Yaskawa INFORM job: X2_8A-21A(90,0).JBI

/JOB
//NAME X2_8A-21A(90,0)
///FOLDERNAME X2
//POS
///NPOS 910,910,910,41,0,0
///TOOL 0
///POSTYPE PULSE
///PULSE
C00000=12667,-135547,-130714,-31270,45596,0
C00001=9315,-159766,-119262,3212,6219,-55552
C00002=157761,-135547,-130714,-31270,45596,69143
C00003=154472,-113934,-104337,-41712,51336,70449
C00004=149832,-108771,-100172,-39130,49259,68869
C00005=148058,-106656,-98467,-38074,48499,68236
C00006=148062,-106275,-96666,-38578,47777,68578
C00007=148058,-106656,-98467,-38074,48499,68236
C00008=147997,-106381,-96958,-38469,47847,68508
C00009=145894,-104035,-96109,-36815,47477,67498
C00010=147997,-106381,-96958,-38469,47847,68508
C00011=154410,-113635,-102825,-42095,50721,70729
C00012=154342,-120637,-107041,-25827,48602,38771
C00013=150292,-111683,-102360,-22573,48994,36710
C00014=148798,-108210,-100464,-21373,49171,35962
C00015=146664,-105787,-99597,-19708,49308,34937
C00016=146949,-106220,-99797,-19932,49282,35074
C00017=147721,-103636,-97533,-20478,49410,35405
C00018=146949,-106220,-99797,-19932,49282,35074
C00019=152261,-118724,-106469,-24248,48548,37770
C00020=148295,-114597,-117137,6490,60568,69086
C00021=147868,-109631,-111600,6790,59752,68875
C00022=147704,-107727,-109395,6911,59390,68790
C00023=147708,-107860,-107783,6984,58336,68724
C00024=147704,-107727,-109395,6911,59390,68790
C00025=147723,-107760,-107968,6963,58499,68740
C00026=147306,-102596,-106094,7098,60024,68678
C00027=147723,-107760,-107968,6963,58499,68740
C00028=148315,-114751,-115749,6537,59639,69038
C00029=148355,-114889,-117236,6461,60467,69101
C00030=147925,-109892,-111692,6763,59663,68890
C00031=147761,-107977,-109485,6884,59305,68805
C00032=147764,-108104,-107870,6957,58254,68739
C00033=147777,-108153,-108078,6942,58354,68751
C00034=147358,-102980,-106206,7078,59886,68688
C00035=147777,-108153,-108078,6942,58354,68751
C00036=148373,-115211,-115873,6515,59468,69049
C00037=147696,-122269,-111871,35505,39043,51945
C00038=147690,-118447,-100224,39719,34874,49579
C00039=148491,-109409,-94254,38171,35277,50420
C00040=148787,-105724,-91002,38010,35060,50504
C00041=148789,-105382,-89977,38411,34697,50285
C00042=149058,-101689,-89016,37046,35623,51030
C00043=149145,-100783,-88679,36755,35795,51189
C00044=149058,-101689,-89016,37046,35623,51030
C00045=145777,-99657,-88811,39022,37803,49998
C00046=148139,-100407,-89095,37251,36591,50936
C00047=145777,-99657,-88811,39022,37803,49998
C00048=147690,-118447,-100224,39719,34874,49579
C00049=128033,-128545,-103748,39689,32513,43973
C00050=128383,-118409,-97778,37905,33566,44930
C00051=128511,-114277,-94563,37658,33626,45064
C00052=128512,-113804,-93446,38069,33271,44843
C00053=129119,-111006,-93029,36452,33958,45715
C00054=129434,-109852,-92636,35862,34111,46033
C00055=128358,-113721,-93936,37885,33613,44941
C00056=176216,-70111,-78093,-55162,70856,80763
C00057=174311,-70781,-78417,-54616,69674,80426
C00058=176216,-70111,-78093,-55162,70856,80763
C00059=181747,-69996,-81392,-56304,75271,81045
C00060=178033,-77165,-93769,-42680,75059,77098
C00061=164745,-109340,-116699,3009,62053,68278
C00062=145851,-112599,-102075,47717,41998,56322
C00063=148044,-104803,-96379,45883,41204,57334
C00064=148864,-101708,-93474,45490,40644,57533
C00065=148866,-101457,-92299,45986,40221,57239
C00066=148863,-101834,-94104,45225,40876,57690
C00067=145127,-99228,-91361,47944,42572,56214
C00068=147466,-100038,-91670,46636,41186,56907
C00069=145127,-99228,-91361,47944,42572,56214
C00070=146129,-107372,-95667,48598,40993,55782
C00071=148216,-109089,-93488,49289,38371,55335
C00072=148344,-107837,-93052,48851,38553,55585
C00073=147906,-112054,-94498,50363,37947,54724
C00074=145851,-112599,-102075,47717,41998,56322
C00075=158250,-140903,-124067,47621,67451,49320
C00076=161740,-133075,-117656,46661,65672,50232
C00077=162335,-130592,-114553,46699,64919,50156
C00078=162276,-129951,-113381,46845,64676,49998
C00079=160420,-132544,-115533,47350,65644,49520
C00080=135901,-74424,-73697,74364,100921,31256
C00081=137788,-75503,-74147,74218,99532,31324
C00082=138769,-76027,-74362,74146,98812,31363
C00083=135901,-74424,-73697,74364,100921,31256
C00084=149282,-147643,-98518,79858,51263,26133
C00085=149394,-146891,-98381,79629,51249,26315
C00086=148448,-152811,-99407,81432,51428,24854
C00087=139735,-166147,-105854,82069,56849,22658
C00088=180438,-97574,-115199,33764,102267,-52414
C00089=189965,-108899,-115705,31971,94091,-51156
C00090=189186,-107218,-114531,32087,94499,-51341
C00091=189186,-107583,-113435,32037,93763,-51550
C00092=190629,-109833,-115910,31859,93547,-51055
C00093=186867,-102382,-113240,32521,96788,-51574
C00094=187005,-102964,-110979,32373,95300,-51952
C00095=188888,-106610,-112304,32065,93703,-51681
C00096=187005,-102964,-110979,32373,95300,-51952
C00097=188021,-107681,-112675,32159,93748,-52003
C00098=189590,-103281,-111094,32025,94271,-51250
C00099=188021,-107681,-112675,32159,93748,-52003
C00100=180438,-97574,-115199,33764,102267,-52414
C00101=185735,-83978,-109774,33564,103394,-50026
C00102=199988,-77820,-108712,-11582,98175,38155
C00103=204749,-56978,-92496,-29836,109182,47433
C00104=202460,-56662,-91339,-29422,107990,46925
C00105=201413,-57385,-91726,-29256,107546,46663
C00106=201611,-57041,-91542,-29296,107663,46703
C00107=201611,-58240,-90431,-29070,106521,47008
C00108=203359,-50274,-87822,-29763,109247,46906
C00109=195470,-25798,-72981,-29209,109868,43903
C00110=195013,-27562,-73704,-29036,109327,43888
C00111=194283,-28250,-74172,-28893,109053,43704
C00112=194480,-28066,-74047,-28932,109127,43754
C00113=194480,-29296,-73135,-28708,108075,44034
C00114=195605,-24849,-71507,-29147,109538,44038
C00115=191110,-5546,-57842,-28597,109561,42465
C00116=192519,-3768,-54500,-33008,111368,41387
C00117=191992,-5303,-55742,-32912,111174,41254
C00118=192059,-5108,-55586,-32924,111198,41271
C00119=192059,-6294,-54683,-32651,110210,41583
C00120=192882,-2296,-53893,-33162,111810,41382
C00121=203365,-15491,-64400,-34648,115083,44256
C00122=218411,-26661,-75493,-58573,107247,46176
C00123=145332,-87800,-123084,-4045,108310,-15756
C00124=109199,-104290,-129101,21867,105305,-43874
C00125=112610,-115777,-129409,14908,94573,-36374
C00126=117115,-112620,-124614,14006,92529,-35127
C00127=118008,-112320,-123068,13816,91609,-34934
C00128=118007,-112900,-122267,13806,90840,-35020
C00129=118044,-112536,-122505,13803,91159,-34973
C00130=118576,-105776,-120168,13731,93052,-34586
C00131=118044,-112536,-122505,13803,91159,-34973
C00132=125955,-111499,-122045,12179,90192,-32457
C00133=127333,-111877,-122174,11884,89885,-32033
C00134=124755,-111115,-121914,12435,90480,-32824
C00135=119624,-116552,-128230,13509,92325,-34321
C00136=117231,-121833,-124467,22052,85463,-28755
C00137=122341,-114124,-118662,20866,84531,-27121
C00138=123318,-113111,-117155,20643,83910,-26885
C00139=123641,-113323,-116249,20585,83205,-26892
C00140=123595,-112804,-116375,20585,83540,-26851
C00141=123397,-106736,-114247,20589,85286,-26623
C00142=123595,-112804,-116375,20585,83540,-26851
C00143=116023,-114044,-115764,22346,84523,-29358
C00144=117346,-116777,-115957,22098,82979,-29171
C00145=118867,-116723,-116143,21757,82713,-28674
C00146=116293,-116772,-115815,22329,83179,-29512
C00147=117231,-121833,-124467,22052,85463,-28755
C00148=154726,-134692,-133300,-19029,79240,-32627
C00149=155157,-123239,-125350,-19102,80279,-32639
C00150=155214,-122106,-123677,-19140,79867,-32554
C00151=155216,-122330,-122794,-19175,79245,-32454
C00152=155272,-122641,-123186,-19186,79334,-32449
C00153=154565,-115790,-120970,-18882,81218,-32994
C00154=155272,-122449,-123985,-19155,79894,-32538
C00155=110972,-119209,-121408,15853,79302,-48266
C00156=109086,-133769,-122042,16854,72857,-49812
C00157=111848,-135958,-122676,16103,71595,-48979
C00158=109086,-133769,-122042,16854,72857,-49812
C00159=108592,-130707,-130810,16554,79646,-49045
C00160=120610,-122471,-119242,21572,81234,-22537
C00161=120610,-122484,-118172,21604,80613,-22649
C00162=120610,-122391,-116483,21658,79689,-22817
C00163=120610,-122419,-116833,21647,79876,-22783
C00164=120610,-122423,-116832,21647,79874,-22783
C00165=120610,-122419,-116833,21647,79876,-22783
C00166=120610,-122416,-116761,21649,79836,-22790
C00167=120610,-122436,-116768,21650,79830,-22791
C00168=120610,-122416,-116761,21649,79836,-22790
C00169=120611,-122370,-120508,21535,82009,-22397
C00170=120611,-120494,-126735,3133,87635,-4471
C00171=120611,-121772,-123926,3138,85252,-4531
C00172=120611,-122092,-122744,3141,84362,-4553
C00173=120611,-122362,-121169,3146,83256,-4581
C00174=120611,-122286,-121724,3144,83636,-4571
C00175=120611,-122290,-121724,3144,83633,-4571
C00176=120611,-122286,-121724,3144,83636,-4571
C00177=120611,-121006,-125813,3134,86805,-4492
C00178=120621,-120378,-125991,12397,109990,-35253
C00179=136832,-143297,-133894,19017,104291,-40845
C00180=187686,-122249,-118318,34521,102174,-42234
C00181=187703,-122088,-115580,34298,100833,-42653
C00182=187707,-122010,-114917,34250,100525,-42749
C00183=187713,-121734,-113169,34135,99743,-42991
C00184=187707,-122010,-114917,34250,100525,-42749
C00185=187770,-121697,-112491,32279,113674,-44764
C00186=187767,-121692,-112491,32279,113678,-44765
C00187=187770,-121697,-112491,32279,113674,-44764
C00188=187667,-121438,-112064,34928,84963,-41689
C00189=187673,-121448,-112068,34927,84958,-41688
C00190=187667,-121438,-112064,34928,84963,-41689
C00191=187641,-121957,-115421,34884,86463,-41227
C00192=173591,-141106,-131528,9997,106250,-69327
C00193=160878,-120510,-126471,37,121976,-81968
C00194=160881,-121699,-123664,37,119637,-81967
C00195=160883,-121991,-122485,37,118762,-81967
C00196=160886,-122244,-120905,37,117660,-81966
C00197=160884,-122111,-121864,37,118318,-81967
C00198=160882,-122100,-121862,36,118322,-81968
C00199=160884,-122111,-121864,37,118318,-81967
C00200=160879,-120821,-125908,37,121469,-81968
C00201=160879,-120821,-131564,37,121469,-81968
C00202=126581,-129511,-133446,-8167,112012,-37796
C00203=82387,-124374,-130385,-21792,102809,55833
C00204=37550,-124758,-124791,-27166,84975,54517
C00205=35933,-124831,-122904,-26864,83389,54284
C00206=35589,-124875,-121597,-26827,82538,54351
C00207=35584,-124889,-121174,-26839,82296,54405
C00208=35764,-126387,-121953,-26892,82093,54519
C00209=31633,-125451,-121673,-25972,81076,53208
C00210=35764,-126387,-121953,-26892,82093,54519
C00211=46981,-157328,-126723,-35790,81436,33730
C00212=42905,-153934,-122174,-35701,78867,32870
C00213=42758,-143813,-119569,-35389,81762,31868
C00214=42905,-153934,-122174,-35701,78867,32870
C00215=53188,-117519,-120731,-36414,97747,30962
C00216=95179,-109851,-129540,-3422,106316,-17944
C00217=143691,-100776,-119079,26047,122130,-73021
C00218=146029,-112499,-120098,24937,116556,-73463
C00219=147204,-116618,-119576,24569,113992,-73590
C00220=147487,-116577,-118677,24502,113425,-73607
C00221=146967,-116625,-120319,24630,114475,-73574
C00222=147345,-121113,-121824,24401,113105,-73737
C00223=146899,-128254,-123879,23878,111030,-74376
C00224=147345,-121113,-121824,24401,113105,-73737
C00225=118081,-135478,-120686,30293,109901,-65237
C00226=118366,-136707,-118609,29972,108136,-65614
C00227=120887,-140213,-119894,30302,106351,-65070
C00228=118366,-136707,-118609,29972,108136,-65614
C00229=117820,-130449,-123242,31209,113594,-64262
C00230=93926,-103398,-125362,18301,106221,-39936
C00231=72688,-110808,-124077,7134,85250,-24096
C00232=75848,-101444,-116923,6191,85411,-23073
C00233=76170,-100985,-115528,6097,84767,-23002
C00234=76167,-101481,-114835,6104,84090,-23035
C00235=78739,-96930,-113773,5320,85595,-22140
C00236=79843,-95445,-113201,4985,85938,-21775
C00237=77748,-98228,-114268,5620,85298,-22470
C00238=140085,-104632,-109249,-40944,98797,6712
C00239=140263,-103640,-106572,-40817,98007,7102
C00240=137942,-102173,-106029,-40697,97269,6378
C00241=140263,-103640,-106572,-40817,98007,7102
C00242=135988,-101428,-112112,-41019,99549,4631
C00243=141957,-83285,-117139,-12315,91699,-6710
C00244=161957,-129781,-122866,20018,67926,-12328
C00245=166016,-109699,-113650,17211,72980,-10098
C00246=174100,-97120,-111511,8065,80457,-7455
C00247=174100,-97549,-110790,8078,79799,-7498
C00248=162725,-116093,-113629,19548,69016,-11850
C00249=162651,-107484,-110669,19284,71494,-11460
C00250=162725,-116093,-113629,19548,69016,-11850
C00251=155151,-112727,-112486,22270,71877,-14160
C00252=155120,-113819,-110277,22518,70103,-14518
C00253=159000,-114269,-110433,21107,68960,-13264
C00254=155120,-113819,-110277,22518,70103,-14518
C00255=155137,-138999,-124748,23105,66364,-15269
C00256=81055,-115973,-127517,-23586,109336,64560
C00257=76492,-127739,-126040,-22738,101683,64421
C00258=76072,-128597,-125529,-22671,100870,64425
C00259=76065,-128640,-125326,-22657,100732,64448
C00260=76072,-128576,-125785,-22685,101025,64394
C00261=82641,-146978,-130130,-22016,96499,67668
C00262=81130,-155003,-132256,-21951,93476,67670
C00263=82641,-146978,-130130,-22016,96499,67668
C00264=84000,-144678,-127518,-21929,96467,68175
C00265=84000,-143983,-126065,-21900,95967,68269
C00266=83327,-146231,-127404,-21916,95478,68108
C00267=88356,-135439,-132684,-22407,104994,68175
C00268=104080,-128245,-132212,31995,84146,22143
C00269=106783,-105266,-117364,31197,85468,23533
C00270=107129,-103609,-115494,31111,85090,23558
C00271=107127,-104217,-114421,31144,84251,23329
C00272=107044,-104571,-114816,31164,84333,23320
C00273=107880,-99055,-112779,30885,85404,23924
C00274=107044,-104571,-114816,31164,84333,23320
C00275=105114,-115284,-123193,31689,84721,22698
C00276=105208,-113465,-123990,31624,85910,23065
C00277=106823,-104635,-117017,31184,85549,23570
C00278=107122,-103295,-115264,31113,85109,23561
C00279=107121,-103855,-114286,31142,84342,23351
C00280=107087,-104437,-114776,31151,84356,23343
C00281=107921,-98925,-112738,30873,85426,23945
C00282=107087,-104437,-114776,31151,84356,23343
C00283=105701,-116384,-125830,31502,85418,23114
C00284=79137,-116524,-127291,7118,77084,-38210
C00285=66518,-158449,-133200,8588,59166,-50817
C00286=70166,-147728,-127011,6864,60501,-49298
C00287=71549,-143558,-123868,6244,60595,-48757
C00288=71544,-142942,-122687,6271,60188,-48782
C00289=71412,-140542,-122600,6259,61371,-48766
C00290=74130,-137647,-121783,5023,62161,-47690
C00291=71412,-140542,-122600,6259,61371,-48766
C00292=59221,-85077,-106862,19044,97138,-55247
C00293=59772,-90133,-108950,18878,95774,-55276
C00294=59221,-85077,-106862,19044,97138,-55247
C00295=65406,-128676,-128270,8670,80773,-42177
C00296=57064,-112054,-129147,2862,108793,-29097
C00297=70948,-123089,-127271,-10962,111372,380
C00298=67644,-116564,-123033,-11394,111660,-848
C00299=67644,-116773,-122597,-11361,111292,-811
C00300=67644,-116291,-123546,-11437,112109,-893
C00301=70770,-123262,-125779,-10903,110357,412
C00302=70770,-123588,-124717,-10837,109552,488
C00303=69306,-120453,-123728,-11077,110342,-115
C00304=70770,-123283,-125719,-10898,110311,416
C00305=70770,-119886,-130778,-11344,115083,-53
C00306=68413,-122856,-123349,-22437,117236,-58
C00307=67404,-122631,-120786,-22344,115611,-123
C00308=67401,-122683,-120099,-22253,115193,-37
C00309=67283,-122594,-120333,-22317,115338,-115
C00310=65261,-118175,-118917,-23034,116088,-1096
C00311=67283,-122594,-120333,-22317,115338,-115
C00312=70820,-123560,-126018,-22187,119059,540
C00313=59587,-128850,-129971,18356,103459,-48793
C00314=60648,-112549,-116046,37363,97913,-74718
C00315=66648,-121539,-115269,36526,91263,-74498
C00316=69624,-125916,-115212,36242,88151,-74300
C00317=69624,-125773,-114639,36242,87924,-74374
C00318=69624,-125814,-114800,36242,87987,-74354
C00319=70738,-127677,-115368,36152,87024,-74211
C00320=69624,-125814,-114800,36242,87987,-74354
C00321=61556,-115340,-115782,37136,96245,-74919
C00322=93863,-107857,-129738,18786,98098,-27923
C00323=113340,-105978,-120535,17383,92037,-15860
C00324=116256,-99504,-115214,16745,91512,-14962
C00325=117368,-96349,-112830,16498,91448,-14602
C00326=124110,-105862,-116355,14920,87592,-12850
C00327=123019,-109757,-118902,15179,87365,-13243
C00328=120254,-118381,-124729,15823,87055,-14212
C00329=121076,-118719,-112405,41381,81563,-9211
C00330=125328,-110839,-107644,40465,80446,-7775
C00331=126920,-107772,-105722,40091,80023,-7243
C00332=122279,-105715,-102241,45382,81605,-7865
C00333=118123,-103314,-98388,50429,83325,-8212
C00334=115452,-99808,-95169,50805,84680,-8860
C00335=113598,-101964,-96694,51043,85596,-9323
C00336=108732,-107177,-100380,51565,88044,-10518
C00337=131658,-113091,-133069,11905,90618,13395
C00338=155934,-143784,-122811,-23124,58745,32427
C00339=151507,-132468,-117411,-20635,59886,30339
C00340=149737,-127499,-115047,-19621,60487,29505
C00341=150974,-127120,-113945,-20271,60326,30034
C00342=146761,-119981,-113829,-13608,66130,25810
C00343=142764,-110481,-112442,-7952,73230,22073
C00344=143750,-114926,-115045,-8343,72653,22456
C00345=146492,-125018,-121022,-9420,71459,23506
C00346=146459,-122334,-129315,-9145,77857,23007
C00347=118526,-115013,-133262,-8809,105739,46794
C00348=93674,-118800,-129721,-8134,120991,68616
C00349=93669,-120967,-127104,-7892,118292,68817
C00350=93667,-121558,-126026,-7814,117333,68886
C00351=93663,-121536,-126144,-7822,117416,68879
C00352=93639,-121762,-126135,-7818,117296,68878
C00353=93680,-121434,-126040,-7817,117406,68885
C00354=93660,-121042,-127131,-7893,118270,68815
C00355=93665,-118880,-129750,-8134,120967,68614
C00356=98446,-113408,-116165,-41475,93741,73013
C00357=93996,-117843,-114815,-40802,89312,72817
C00358=91343,-117266,-113836,-40455,87860,72224
C00359=92137,-119395,-114109,-40564,87510,72703
C00360=95072,-126184,-113786,-40951,86041,74561
C00361=95071,-125918,-112907,-40977,85731,74679
C00362=96936,-125131,-114749,-41104,87782,74702
C00363=101504,-121000,-116278,-41571,92256,74948
C00364=100864,-122088,-112493,-43204,76282,71688
C00365=95643,-121963,-109784,-42340,72556,70846
C00366=93677,-120964,-108398,-41948,71358,70433
C00367=93599,-121011,-107366,-42074,70823,70622
C00368=95642,-121622,-108630,-42447,72155,71017
C00369=100864,-121830,-111367,-43291,75868,71867
C00370=131033,-115476,-133015,-2815,101744,74384
C00371=151471,-119125,-123137,34971,103386,73225
C00372=162012,-101235,-114016,37763,108592,75954
C00373=163745,-105512,-114443,37294,106318,75861
C00374=162987,-105303,-114126,37291,106564,75626
C00375=159264,-105978,-111996,36953,106780,74110
C00376=157962,-101866,-111865,37402,108959,74341
C00377=155898,-93647,-112180,38609,113341,75115
C00378=179206,-139250,-107986,62075,77828,66561
C00379=185232,-138953,-105140,62379,73225,66913
C00380=188358,-139601,-104691,62502,70946,67188
C00381=188182,-138293,-102809,62647,70826,66949
C00382=185238,-138055,-103864,62461,73065,66778
C00383=179211,-138396,-106727,62132,77661,66424
C00384=179188,-148562,-121526,61524,79591,68010
C00385=184417,-115822,-131978,19629,107310,-7500
C00386=190427,-134899,-136820,-8574,116374,-78562
C00387=188066,-120573,-128029,-9218,118052,-79593
C00388=191728,-147691,-136467,-6881,103686,-75134
C00389=187922,-120139,-126444,-9176,117292,-79584
C00390=187907,-121816,-124776,2981,114509,-78147
C00391=187942,-121398,-126015,3016,115485,-78109
C00392=187937,-119495,-128851,3098,118205,-78035
C00393=176042,-128909,-129640,7380,110692,-58022
C00394=187833,-113452,-115854,34994,105139,-41767
C00395=187847,-113781,-113588,34722,103839,-42187
C00396=187853,-113844,-112659,34623,103335,-42348
C00397=187856,-113866,-111596,34519,102780,-42525
C00398=187851,-113844,-112538,34611,103274,-42368
C00399=187836,-113627,-114840,34866,104547,-41960
C00400=186756,-108501,-120882,36201,110201,-40487
C00401=150585,-129060,-123753,46684,114085,39870
C00402=134046,-137019,-115206,49635,112096,74674
C00403=134033,-140586,-110307,48065,108843,72866
C00404=134037,-138671,-107458,47843,108316,72589
C00405=133982,-137493,-106313,47802,108278,72540
C00406=134018,-151682,-126528,-1136,113553,57560
C00407=134015,-151576,-126422,-1136,113542,57558
C00408=134097,-144792,-115626,-40459,90065,47115
C00409=134072,-145102,-116392,-40468,90292,47016
C00410=134074,-146851,-118858,-40485,90771,46834
C00411=141855,-151854,-132376,-33568,89282,32323
C00412=173958,-148748,-133240,-11874,65312,-15203
C00413=187653,-128002,-123664,7056,57779,-46476
C00414=188071,-112180,-99768,-1790,31671,-46486
C00415=188092,-111455,-97340,-1875,30550,-46442
C00416=187648,-111286,-97015,-1307,30429,-46727
C00417=187657,-110013,-93933,-1370,29188,-46699
C00418=187545,-109794,-93383,-1224,28959,-46769
C00419=187645,-108907,-90946,-1403,27919,-46677
C00420=188106,-109627,-92159,-2030,28303,-46362
C00421=188086,-110531,-94662,-1935,29378,-46411
C00422=188086,-114129,-114927,-1479,39995,-46659
C00423=201470,-41376,-102585,-19941,97743,57993
C00424=197439,-2624,-49840,-39121,107911,51008
C00425=168391,92926,48790,-27485,116767,48744
C00426=170067,83268,36769,-27957,119460,48700
C00427=172466,59632,8553,-30739,114348,38093
C00428=173361,44257,-8636,-31524,116948,37644
C00429=173383,42327,-10579,-31793,119746,39948
C00430=177083,19842,-31222,-36073,117787,44685
C00431=167208,60082,10679,-34630,117458,49250
C00432=186843,33187,-28183,-45340,118495,56566
C00433=187270,22965,-40018,-42118,113549,44205
C00434=164927,12374,-50848,-37497,97302,-26684
C00435=160848,-52651,-98971,-6904,73590,-44156
C00436=187933,-111679,-98706,278,30585,-46526
C00437=187953,-110958,-96368,260,29517,-46517
C00438=187785,-110792,-95734,491,29212,-46632
C00439=187759,-109968,-93159,543,28049,-46662
C00440=187728,-109749,-92348,600,27665,-46686
C00441=187829,-108748,-90356,464,26951,-46620
C00442=187968,-109087,-91174,258,27282,-46516
C00443=187948,-109974,-93584,278,28309,-46526
C00444=190713,-138118,-122139,-3147,45685,-54861
C00445=188097,-104568,-127563,-3199,90457,-72619
C00446=188112,-108983,-124849,-3203,86524,-72515
C00447=195921,-129294,-127631,-11282,74318,-69986
C00448=192645,-118053,-125281,-7801,80438,-71273
C00449=186991,-123845,-126852,-2601,76931,-72588
C00450=191356,-129057,-127829,-6636,73864,-71242
C00451=188153,-109076,-124888,-3215,86502,-72501
C00452=188138,-104664,-127604,-3212,90434,-72606
C00453=187898,-111965,-120493,16766,69565,-69566
C00454=187918,-113285,-117348,17044,67055,-69927
C00455=188130,-114919,-116177,17134,65516,-70081
C00456=187738,-112085,-115217,17212,66427,-70088
C00457=187693,-112142,-115274,17234,66443,-70102
C00458=187708,-111963,-115192,17225,66482,-70091
C00459=187944,-113344,-117352,17035,67023,-69922
C00460=187924,-112030,-120500,16757,69531,-69561
C00461=180038,-109975,-126789,2440,82512,7441
C00462=174468,-102021,-118148,1871,82653,17547
C00463=174479,-103807,-115834,1877,80312,17516
C00464=175222,-104980,-115127,1627,79258,17743
C00465=175101,-105254,-115206,1669,79168,17704
C00466=174304,-107092,-109423,11728,69502,18325
C00467=172906,-107949,-109483,12341,69309,17805
C00468=174390,-105691,-110273,11607,70709,18474
C00469=174377,-104937,-112785,11492,72607,18653
C00470=190845,-100837,-124447,-13698,93294,33124
C00471=206306,-116062,-120388,-37359,88631,50073
C00472=215039,-120395,-106715,-50971,83253,62053
C00473=215038,-119729,-104733,-51036,82687,62365
C00474=215491,-118695,-103696,-51084,82872,62503
C00475=215838,-117471,-101038,-51193,82418,62940
C00476=215047,-118800,-102176,-51129,81987,62759
C00477=215049,-119543,-104187,-51057,82539,62453
C00478=215012,-122438,-115563,-50746,86080,60488
C00479=160845,-113405,-113287,-47121,77099,-31472
C00480=160851,-113463,-110064,-47446,75709,-30781
C00481=159953,-113580,-108952,-47357,74728,-30737
C00482=160713,-112885,-108716,-47509,75268,-30630
C00483=160788,-113231,-109982,-47419,75724,-30819
C00484=160782,-112987,-114684,-46949,77813,-31850
C00485=161690,-87231,-108001,-36248,90547,-80444
C00486=156808,-90580,-101865,-35022,84112,-80274
C00487=153093,-73717,-94488,-33864,86116,-82332
C00488=158330,-83683,-104653,-35339,89043,-81248
C00489=160758,-112853,-114863,-36163,82877,-78288
C00490=160760,-113152,-111426,-36317,81029,-77674
C00491=159972,-107251,-112602,-31595,97855,-78366
C00492=161125,-112629,-114388,-31534,96843,-77635
C00493=163818,-123639,-118907,-29284,98848,-76882
C00494=165784,-130773,-121304,-28132,99036,-76085
C00495=160757,-112482,-116558,-30024,102576,-77779
C00496=160755,-111254,-119690,-30396,104801,-78387
C00497=139139,-104942,-132434,-5076,105021,-81413
C00498=120610,-140892,-128239,26796,83300,-73925
C00499=124485,-139346,-124335,26282,80622,-73071
C00500=130128,-175956,-130442,27969,57436,-76413
C00501=124992,-173069,-127473,33175,56379,-79351
C00502=128349,-154705,-122706,28450,56573,-77464
C00503=139577,-169309,-125107,18432,42001,-69520
C00504=128860,-155984,-126780,25446,58633,-74277
C00505=138109,-135032,-133743,8289,74304,-51513
C00506=203654,-125968,-124215,-37381,73551,30645
C00507=201127,-103516,-110680,-20461,62884,59060
C00508=201138,-104157,-107983,-20829,61019,59420
C00509=202030,-104808,-106563,-21546,60112,59957
C00510=202002,-105410,-106700,-21580,59897,59992
C00511=201699,-105782,-106630,-21465,59600,59928
C00512=201116,-104130,-107973,-20816,61021,59411
C00513=201105,-103488,-110669,-20449,62886,59051
C00514=198523,-119273,-121454,-24683,77158,64296
C00515=174403,-100049,-121231,-21877,99309,62114
C00516=174406,-102879,-118773,-21681,96545,62622
C00517=173414,-104710,-118266,-21449,95131,62534
C00518=174393,-105461,-115937,-21537,93676,63134
C00519=174418,-104205,-117181,-21599,94999,62906
C00520=174415,-101880,-119808,-21752,97619,62429
C00521=185776,-93152,-118465,1785,83350,67432
C00522=169060,-142396,-123848,37084,49654,60484
C00523=174230,-113472,-108308,34615,49911,64397
C00524=174247,-112967,-104740,35556,48304,63744
C00525=175666,-113779,-103346,35329,46667,63822
C00526=175539,-113458,-102511,35603,46435,63646
C00527=175333,-116338,-102041,36740,45079,62916
C00528=175333,-116330,-102018,36746,45071,62912
C00529=175687,-114680,-100844,36447,45022,63094
C00530=186215,-128372,-100068,26026,26198,70682
C00531=176941,-119437,-104065,35607,43539,63699
C00532=174229,-113129,-105847,35265,48804,63944
C00533=182962,-136134,-123657,29797,44727,67038
C00534=210827,-121899,-127370,35396,86436,76908
C00535=214505,-124636,-123608,35577,86411,76994
C00536=214521,-124823,-120077,35640,84542,76397
C00537=211296,-135461,-118635,40120,76829,77549
C00538=217173,-131905,-117674,36934,71435,81853
C00539=214545,-124844,-120083,35636,84527,76402
C00540=214528,-124659,-123615,35573,86395,76999
C00541=214596,-124890,-121786,39550,96156,78039
C00542=214607,-124784,-118461,39383,94595,77461
C00543=216868,-117162,-114438,39473,95627,77942
C00544=216826,-117733,-111908,39235,93442,77833
C00545=214785,-119888,-114308,39371,94481,77497
C00546=214619,-124823,-118761,39395,94718,77513
C00547=214540,-124430,-116246,48349,86426,68042
C00548=214499,-123956,-126099,48385,90728,70182
C00549=158797,-145907,-128305,56145,74291,56792
C00550=118138,-117595,-113507,59219,64127,52420
C00551=134091,-119062,-102284,58108,50235,52331
C00552=134095,-117716,-98836,59129,49460,51612
C00553=136880,-117696,-97684,58682,47369,51919
C00554=134362,-122362,-110313,11427,42979,62451
C00555=135446,-122601,-110257,10536,42675,62953
C00556=134922,-122649,-109830,10807,42225,63366
C00557=135201,-122130,-106007,7130,38171,71932
C00558=134097,-120880,-107281,7954,39689,71484
C00559=133538,-122024,-122159,7272,48238,71950
C00560=134045,-120979,-109361,39707,45136,55893
C00561=134048,-117179,-98466,43015,41514,53843
C00562=135089,-118697,-98895,40257,39934,54577
C00563=134334,-118944,-102166,12845,37385,61615
C00564=134107,-119314,-102576,13047,37486,61499
C00565=123808,-118793,-97951,-36574,37979,75667
C00566=134076,-115553,-94209,-55177,43841,79182
C00567=133651,-114033,-99266,-51853,45977,77066
C00568=134816,-132236,-131789,6177,48808,72548
C00569=152519,-98596,-126841,17039,86437,59409
C00570=167034,-82548,-116958,26153,108191,47353
C00571=167227,-85698,-113927,25595,104988,46679
C00572=151895,-76409,-102172,41212,110118,45490
C00573=159565,-75916,-103746,36963,107071,46708
C00574=168155,-63475,-98008,36210,106114,49753
C00575=170878,-58988,-95708,35874,105831,50700
C00576=180979,-58723,-101497,23976,107062,51805
C00577=180909,-54943,-104050,24554,110296,52487
C00578=168157,-75412,-102271,33648,91006,21456
C00579=174012,-67106,-91297,33471,82630,14810
C00580=175466,-61382,-85667,32996,81659,15067
C00581=175951,-59606,-83647,32846,81204,15115
C00582=202871,-62360,-90085,-4336,78171,36795
C00583=160162,-88082,-101553,14242,74573,22768
C00584=153958,-94067,-102293,19502,70417,24299
C00585=154362,-96202,-104591,19297,70625,24481
C00586=154503,-104813,-110762,19306,69999,24428
C00587=155575,-73729,-96860,32555,86012,14938
C00588=157088,-68154,-91284,32096,84992,15206
C00589=157307,-67802,-89787,32053,84283,15086
C00590=177382,-78627,-97768,6885,75030,28579
C00591=165969,-82047,-99209,11770,75418,24820
C00592=194698,-86953,-95499,-27526,68480,52539
C00593=201423,-82172,-92479,-35779,72324,57601
C00594=205660,-83542,-95477,-37134,74990,58446
C00595=150225,-90058,-124320,20069,81923,14603
C00596=88917,-116100,-126028,29630,66347,-39612
C00597=48102,-114880,-112674,35477,56596,-75725
C00598=53396,-105773,-101201,33500,52497,-74682
C00599=53385,-105323,-98106,34230,51099,-75219
C00600=48945,-100827,-95317,40107,56687,-78941
C00601=72663,-108261,-98237,-972,40027,-55342
C00602=53363,-105522,-99057,19217,46878,-60217
C00603=53371,-105892,-101942,18746,48378,-59901
C00604=53322,-113038,-104699,-812,43724,-42660
C00605=53318,-112442,-102021,-830,42382,-42650
C00606=53317,-112163,-100935,-837,41857,-42645
C00607=53253,-112229,-97736,-1547,37461,-42516
C00608=53300,-111445,-98358,-1568,38246,-42506
C00609=51520,-115460,-104005,179,39644,-43460
C00610=55761,-139961,-122674,27476,66843,-55729
C00611=53542,-121644,-113892,40363,83761,-61539
C00612=53523,-121175,-111327,40444,82737,-61941
C00613=53533,-120846,-110023,41635,87424,-59647
C00614=53533,-120798,-109834,41636,87355,-59676
C00615=53529,-120315,-108043,41648,86710,-59935
C00616=53536,-120580,-109029,41640,87063,-59791
C00617=53556,-121151,-111460,41628,87965,-59422
C00618=52633,-122748,-126719,40391,89833,-59612
C00619=140119,-108661,-130674,21165,82789,25459
C00620=161125,-123349,-120158,18581,66270,46079
C00621=161135,-123185,-116439,18891,64175,45732
C00622=161233,-123294,-114830,19012,63160,45595
C00623=161362,-123797,-115013,18974,62993,45618
C00624=163252,-122153,-114536,18047,63094,46376
C00625=161212,-123488,-116538,18871,64068,45743
C00626=161202,-123677,-120265,18562,66156,46089
C00627=167124,-146469,-125858,-32695,63076,70922
C00628=161220,-122264,-110536,-44525,64077,74742
C00629=161219,-121375,-107584,-44985,63095,75224
C00630=164956,-113855,-102560,-48427,66781,75111
C00631=161213,-120936,-106323,-43985,60856,74418
C00632=162410,-115678,-102562,-44623,57414,74861
C00633=159906,-125883,-101158,-48949,49496,78085
C00634=161197,-119682,-102993,-46927,53134,76618
C00635=161197,-120736,-105876,-46275,53998,76117
C00636=161177,-121556,-108554,-35078,57327,43050
C00637=161177,-120932,-106617,-35398,56609,43319
C00638=152937,-127654,-109782,-25136,48983,42100
C00639=161176,-119640,-103030,-36318,54707,44163
C00640=161179,-121241,-107541,-34339,64662,45277
C00641=161179,-121533,-108462,-34233,65010,45160
C00642=161180,-122193,-110741,-33972,65899,44866
C00643=159909,-111206,-128347,10927,59798,43136
C00644=174276,-119239,-128019,-9099,73009,-32604
C00645=174287,-122281,-118814,-9519,65873,-32039
C00646=174304,-122135,-115653,-9666,64029,-31878
C00647=174310,-122046,-114838,-9707,63581,-31838
C00648=174391,-121924,-120589,9734,82175,-37722
C00649=174107,-122717,-120904,9805,81999,-37834
C00650=171570,-123633,-117371,28457,102738,-42839
C00651=174312,-121937,-114098,33622,107981,-42892
C00652=174299,-122214,-116525,33911,109120,-42531
C00653=174287,-119835,-127268,36019,115609,-40290
C00654=15972,-110889,-128286,10965,59905,43045
C00655=15972,-110889,-128286,10965,59905,43045
C00656=53465,-86935,-89811,40465,79071,-68727
C00657=72562,-12745,-29122,31918,77028,-65113
C00658=126847,105220,75143,-13359,85174,-71704
C00659=126692,103863,77460,-13374,83082,-71533
C00660=126630,103456,78567,-13386,82202,-71459
C00661=126630,104061,81025,-13418,81032,-71332
C00662=126630,103456,78567,-13386,82202,-71459
C00663=127186,113222,93196,-13600,78417,-70848
C00664=126835,106827,84700,-13475,80250,-71174
C00665=127186,112337,90806,-13561,79406,-70955
C00666=125466,108208,85326,-13267,80342,-71662
C00667=125456,110134,89113,-13313,79033,-71523
C00668=125851,108129,86455,-13346,79687,-71457
C00669=125851,107524,84502,-13315,80555,-71552
C00670=127397,113852,88268,-13512,81719,-71138
C00671=127478,100573,81223,-12545,72653,-68441
C00672=127453,88829,76924,-10550,63166,-66037
C00673=131548,87777,90621,-11121,47758,-61203
C00674=131548,89037,93025,-11267,46942,-61104
C00675=131184,80149,80924,-10608,49723,-61589
C00676=131184,81034,82789,-10715,49041,-61514
C00677=131266,84902,87812,-10945,47967,-61355
C00678=131383,76857,75341,-10452,51464,-61690
C00679=130781,66873,56355,-9383,57854,-62552
C00680=132527,42070,31553,4220,55444,-80155
C00681=132770,47352,42186,4293,51610,-80213
C00682=132777,48864,44545,4331,50936,-80239
C00683=132777,49184,45555,4359,50481,-80259
C00684=131974,44354,39680,4735,51658,-80551
C00685=131974,44660,40691,4765,51193,-80574
C00686=132343,47526,43917,4586,50669,-80439
C00687=132425,45260,40696,4491,51479,-80364
C00688=131916,38002,29050,4572,54929,-80427
C00689=154349,-2508,-17410,-792,70409,-75613
C00690=173270,57866,35055,-970,89791,-77800
C00691=173007,64123,36896,-949,91868,-77904
C00692=159395,25803,23488,1167,50974,-82636
C00693=159231,31527,34115,1332,47380,-82754
C00694=159081,33176,36534,1437,46744,-82832
C00695=159081,33667,37902,1449,46152,-82839
C00696=159081,33176,36534,1437,46744,-82832
C00697=159294,29405,33293,1303,46796,-82733
C00698=159294,29665,34034,1311,46474,-82739
C00699=159347,31699,36068,1285,46267,-82719
C00700=159294,29665,34034,1311,46474,-82739
C00701=159426,21602,21138,1160,50263,-82632
C00702=180997,48207,44640,-11318,50849,-73280
C00703=180806,54122,56304,-11930,46765,-72867
C00704=180779,55045,58047,-12031,46174,-72803
C00705=180782,56411,61345,-12306,44876,-72626
C00706=180779,55045,58047,-12031,46174,-72803
C00707=181200,49240,53369,-12299,46136,-72602
C00708=180943,52994,57542,-12278,45474,-72631
C00709=181200,49240,53369,-12299,46136,-72602
C00710=181426,42658,40426,-11597,50658,-73068
C00711=124517,-23255,-20984,17957,59356,-58990
C00712=94820,-59465,-69818,28302,74069,-32860
C00713=94820,-59465,-69818,28302,74069,-32860
C00714=97675,-88762,-33594,39297,33668,-1326
C00715=144147,-78557,-16505,-24092,15269,-14703
C00716=130185,7163,36266,2840,25337,-83020
C00717=148170,13776,15406,2916,63739,-81295
C00718=150199,5381,460,4242,84465,-83896
C00719=150319,4565,3801,4247,81990,-83938
C00720=149634,5975,6642,4316,81003,-84208
C00721=149635,6585,8872,4325,79950,-84244
C00722=149634,2811,-12782,4285,91305,-83856
C00723=149753,9380,-6624,4276,90884,-83829
C00724=149753,9452,-5229,4274,90064,-83857
C00725=149716,8162,-6363,4279,90100,-83869
C00726=149896,8565,-6046,4260,90105,-83810
C00727=149739,11202,-9295,4288,93459,-83747
C00728=159769,-26352,-42847,-7626,75430,-42908
C00729=160661,-23608,-37245,-8003,73495,-42476
C00730=160801,-19429,-32426,-8083,72699,-42375
C00731=160801,-19408,-31304,-8110,72027,-42329
C00732=161009,-22449,-34949,-8156,72720,-42303
C00733=160818,-23595,-34308,-8131,71724,-42302
C00734=160891,-21766,-32937,-8155,71827,-42286
C00735=161249,-23550,-34138,-8284,71688,-42148
C00736=159612,-30937,-44211,-7622,73912,-42867
C00737=144117,-44081,-61004,17211,89666,-8724
C00738=145648,-40124,-55468,16926,88039,-8426
C00739=146237,-38515,-53215,16819,87384,-8313
C00740=146244,-38444,-53170,16818,87391,-8310
C00741=146245,-38577,-51594,16825,86395,-8446
C00742=146244,-38444,-53170,16818,87391,-8310
C00743=146240,-38608,-52193,16823,86734,-8401
C00744=146535,-35573,-50236,16765,87015,-8261
C00745=146268,-38521,-51765,16819,86519,-8421
C00746=147801,-39090,-52130,16535,86146,-7942
C00747=146268,-38521,-51765,16819,86519,-8421
C00748=144117,-44081,-61004,17211,89666,-8724
C00749=145162,-56828,-95851,3587,97052,-36303
C00750=147136,-55674,-91646,3015,94990,-35768
C00751=150906,-56103,-90461,1950,93937,-34650
C00752=150909,-57277,-89363,1945,92659,-34669
C00753=150906,-56103,-90461,1950,93937,-34650
C00754=147900,-55107,-89916,2796,94193,-35556
C00755=147871,-56692,-89008,2798,92822,-35595
C00756=149697,-57326,-89351,2285,92656,-35040
C00757=147871,-56692,-89008,2798,92822,-35595
C00758=149264,-52275,-86592,2410,93564,-35155
C00759=149536,-48545,-84471,2336,94168,-35061
C00760=149264,-52275,-86592,2410,93564,-35155
C00761=145162,-56828,-95851,3587,97052,-36303
C00762=148725,-41791,-46801,46253,72923,63254
C00763=150766,-40622,-42529,46203,70442,63063
C00764=151958,-40590,-41445,46071,69368,63137
C00765=152929,-23174,-29921,45352,70192,64025
C00766=151861,-23991,-31407,45521,71087,63922
C00767=150038,-24992,-35653,45558,73508,64179
C00768=157424,-58492,-62688,32217,54755,56547
C00769=158288,-54308,-56839,32290,53193,56420
C00770=158982,-52601,-54844,32035,52629,56561
C00771=163111,-53232,-55421,29606,51160,58075
C00772=162018,-54402,-56899,30142,51809,57760
C00773=161259,-58664,-62788,30049,53328,57890
C00774=162071,-38381,-52824,22779,71448,67723
C00775=155468,-16762,-35985,12938,95334,79413
C00776=155428,-21282,-38074,12915,94327,79293
C00777=155428,-21377,-36350,12890,93245,79180
C00778=158883,-21661,-36555,12572,92691,80303
C00779=158883,-20912,-43127,12689,97018,80745
C00780=156175,-29321,-49040,12925,96764,79803
C00781=147061,-19099,-23009,3757,61390,3418
C00782=130185,-5552,7433,2044,36537,-20417
C00783=151147,-94304,-42406,-24574,24293,-13335
C00784=97675,-114303,-72306,31404,42508,3161
C00785=152316,-10513,-15673,4526,58659,36023
C00786=151393,3749,17430,6351,28873,74416
C00787=149831,7562,23171,8658,27454,73145
C00788=155239,11547,33415,-11686,18033,81661
C00789=150955,12605,34257,-2991,17680,77198
C00790=154914,8269,24071,-18383,27125,83176
C00791=154718,5177,20099,-17644,27899,82791
C00792=167718,25210,36606,30956,40836,49421
C00793=167855,32077,47382,32851,38131,48328
C00794=167909,35118,52103,33773,36979,47811
C00795=169559,35638,52638,32786,36297,48539
C00796=169779,35717,52719,32651,36207,48636
C00797=170327,35923,52931,32313,35983,48881
C00798=170290,32850,48162,31377,37157,49401
C00799=170195,25923,37295,29460,39906,50494
C00800=161814,1273,-11441,3222,75062,5973
C00801=136959,1837,906,-7736,58378,-48926
C00802=124978,70134,45130,-8465,63129,-67393
C00803=125101,72944,51302,-8704,60813,-67169
C00804=125052,50106,45596,-10128,37231,-64881
C00805=121107,58271,54717,-6630,35418,-66921
C00806=121137,36579,27666,-5899,40889,-67339
C00807=125358,93261,79640,-22528,73899,-61469
C00808=125277,100468,81878,-21599,81132,-62849
C00809=125335,101024,83815,-21652,80302,-62678
C00810=124852,92731,73597,-21836,79166,-62649
C00811=124875,90292,70970,-22108,77307,-62299
C00812=120144,99725,81932,-17388,74332,-63487
C00813=120132,119163,106853,-17403,74692,-63545
C00814=119700,121745,110389,-17420,73788,-63569
C00815=117452,89281,65020,-12631,78853,-64898
C00816=109757,84264,56014,2090,83450,-32603
C00817=104431,79702,59666,14857,76182,-33127
C00818=104213,82742,69971,15234,71602,-33782
C00819=108045,71800,59855,7296,68082,-23100
C00820=109903,73729,64230,2381,65624,-17202
C00821=112200,81345,64646,-2754,78368,-12208
C00822=122013,87109,77034,-10739,68212,9471
C00823=122753,87378,74154,-12404,66890,11820
C00824=122931,87850,76379,-12558,65817,12004
C00825=112195,84601,72597,11005,65721,-14617
C00826=112765,82325,69769,10787,66205,-14358
C00827=122948,67196,62583,-5625,62671,-18437
C00828=138903,24520,6015,-29218,77766,-47278
C00829=110595,-133836,-92325,-25734,64127,-40353
C00830=215771,-69947,-53674,-42443,70025,1415
C00831=144700,-70309,-53328,41384,55522,26317
C00832=159027,-8981,-29340,14833,99808,55594
C00833=157462,-4946,-22039,14756,97743,54798
C00834=156376,7564,-8740,18840,102766,55428
C00835=155948,14858,-2592,15200,104674,55259
C00836=156571,-6804,-23527,14776,97863,54502
C00837=156840,-8773,-29171,14894,100200,54881
C00838=162486,-26662,-42491,16083,70936,60571
C00839=162478,-24897,-37244,16311,68704,60258
C00840=169307,-31861,-37755,7343,57905,60976
C00841=166646,-32506,-38185,8784,58103,59938
C00842=159367,-24765,-36916,18592,69259,59149
C00843=159276,-26541,-42171,18380,71485,59471
C00844=144700,-70309,-53328,41384,55522,26317
C00845=199062,-57325,-47228,-38260,64183,-4080
C00846=130069,-136035,-99643,-25251,40054,-29144
C00847=138295,14600,-5239,-29006,77829,-46706
C00848=134460,50083,49848,-7522,47450,-72891
C00849=133863,54044,57016,-7448,45040,-72971
C00850=135329,50298,57934,-10829,38014,-71386
C00851=130984,58940,67136,-7218,37329,-73683
C00852=129992,63475,69286,-5254,42047,-74620
C00853=129939,57134,57748,-4871,45871,-74863
C00854=131463,20221,19829,13252,41381,-77379
C00855=132193,24627,26872,13213,39243,-77340
C00856=133755,26108,29466,12113,38187,-76660
C00857=135940,24164,27686,10218,37980,-75490
C00858=134234,21276,23788,11460,39107,-76261
C00859=134362,17227,17019,10879,41136,-75917
C00860=136755,-1514,-5704,2516,47370,-67254
C00861=146721,-74009,-73220,-16059,57976,-45633
C00862=199062,-57325,-47228,-38260,64183,-4080
C00863=144700,-70309,-53328,41384,55522,26317
C00864=155243,-37029,-47289,14287,81392,50093
C00865=162013,-14853,-33688,-2862,92831,64763
C00866=161094,-16180,-30749,-2749,90312,64514
C00867=150871,-13866,-27733,624,94437,61273
C00868=148787,-16966,-29949,-104,92140,60503
C00869=151795,-16277,-35009,-342,95617,61503
C00870=149948,-19918,-37445,-1443,92226,60777
C00871=164755,-27863,-42732,-4142,59506,66566
C00872=162884,-23098,-35965,-3113,57711,65906
C00873=163814,-21174,-33012,-3697,56921,66298
C00874=160932,-21340,-33244,-1979,56878,65160
C00875=166382,-34706,-48953,-5069,59907,67170
C00876=176106,-57995,-75379,-10186,65060,70407
C00877=133349,-74401,-55247,45018,60413,22671
C00878=199062,-57325,-47228,-38260,64183,-4080
C00879=152753,-113498,-70464,-41238,43505,-17390
C00880=177120,60337,38950,-9482,83637,54876
C00881=178509,86919,73346,-3525,79260,66985
C00882=178771,91754,83117,-3597,75750,67174
C00883=178771,93528,87156,-3622,74179,67221
C00884=174873,87450,79527,-3137,75585,65824
C00885=174873,84343,71196,-3099,79110,65736
C00886=148723,11111,-11073,115,91617,56758
C00887=170148,33267,40244,13523,40602,55072
C00888=169779,39993,51106,14764,37530,54327
C00889=170966,42923,55759,14284,36006,54701
C00890=166085,41238,54012,17998,37157,52177
C00891=165316,38755,49817,18049,38567,52082
C00892=165615,32055,39029,16711,41561,52889
C00893=145399,5848,-6390,-3865,80891,44221
C00894=150200,-72379,-61943,-28480,64443,2945
C00895=199062,-57325,-47228,-38260,64183,-4080
C00896=144700,-70309,-53328,41384,55522,26317
C00897=142540,-54200,-62960,20837,71495,76935
C00898=143745,-53250,-58469,20670,69060,76947
C00899=144539,-52645,-56954,20458,68281,77109
C00900=145328,-36296,-50730,18144,82290,78247
C00901=145614,-29529,-48100,16778,93497,78591
C00902=145614,-29529,-48100,16778,93497,78591
C00903=144903,-28900,-49357,16896,94730,78514
C00904=146283,-22644,-55524,17079,101176,79886
C00905=143098,-32267,-54477,15830,97365,74738
C00906=144038,-90899,-70127,40115,59013,77438
C00907=150229,-119732,-79060,43329,46830,76451
C00908=120872,-104982,-67229,50399,61266,16237
C00909=12667,-135547,-130714,-31270,45596,0
BC00000=78377,519142,1075139
BC00001=177043,462590,1002506
BC00002=78377,276983,1075139
BC00003=70777,286120,1075139
BC00004=70777,286120,1075139
BC00005=70777,286120,1075139
BC00006=70777,286120,1075139
BC00007=70777,286120,1075139
BC00008=70777,286120,1075139
BC00009=70777,286120,1075139
BC00010=70777,286120,1075139
BC00011=70777,286120,1075139
BC00012=103885,292860,1075139
BC00013=103885,292860,1075139
BC00014=103885,292860,1075139
BC00015=103885,292860,1075139
BC00016=103885,292860,1075139
BC00017=103885,292860,1075139
BC00018=103885,292860,1075139
BC00019=103885,292860,1075139
BC00020=89899,279578,1075139
BC00021=89899,279578,1075139
BC00022=89899,279578,1075139
BC00023=89899,279578,1075139
BC00024=89899,279578,1075139
BC00025=89899,279578,1075139
BC00026=89899,279578,1075139
BC00027=89899,279578,1075139
BC00028=89899,279578,1075139
BC00029=27352,290463,1075139
BC00030=27352,290463,1075139
BC00031=27352,290463,1075139
BC00032=27352,290463,1075139
BC00033=27352,290463,1075139
BC00034=27352,290463,1075139
BC00035=27352,290463,1075139
BC00036=27352,290463,1075139
BC00037=160737,417922,1075139
BC00038=160737,417922,1075139
BC00039=160737,417922,1075139
BC00040=160737,417922,1075139
BC00041=160737,417922,1075139
BC00042=160737,417922,1075139
BC00043=160737,417922,1075139
BC00044=160737,417922,1075139
BC00045=160737,417922,1075139
BC00046=160737,417922,1075139
BC00047=160737,417922,1075139
BC00048=160737,417922,1075139
BC00049=123386,424393,1075139
BC00050=123386,424393,1075139
BC00051=123386,424393,1075139
BC00052=123386,424393,1075139
BC00053=123386,424393,1075139
BC00054=123386,424393,1075139
BC00055=123386,424393,1075139
BC00056=123386,424393,1075139
BC00057=123386,424393,1075139
BC00058=123386,424393,1075139
BC00059=123386,424393,1075139
BC00060=129448,421831,1075139
BC00061=151133,412666,1075139
BC00062=169673,404485,1075139
BC00063=169673,404485,1075139
BC00064=169673,404485,1075139
BC00065=169673,404485,1075139
BC00066=169673,404485,1075139
BC00067=169673,404485,1075139
BC00068=169673,404485,1075139
BC00069=169673,404485,1075139
BC00070=169673,404485,1075139
BC00071=169673,404485,1075139
BC00072=169673,404485,1075139
BC00073=169673,404485,1075139
BC00074=169673,404485,1075139
BC00075=120098,376458,1075139
BC00076=120098,376458,1075139
BC00077=120098,376458,1075139
BC00078=120098,376458,1075139
BC00079=120098,376458,1075139
BC00080=120098,376458,1075139
BC00081=120098,376458,1075139
BC00082=120098,376458,1075139
BC00083=120098,376458,1075139
BC00084=120098,376458,1075139
BC00085=120098,376458,1075139
BC00086=120098,376458,1075139
BC00087=120098,376458,1075139
BC00088=141865,351941,1075139
BC00089=141865,351941,1075139
BC00090=141865,351941,1075139
BC00091=141865,351941,1075139
BC00092=141865,351941,1075139
BC00093=141865,351941,1075139
BC00094=141865,351941,1075139
BC00095=141865,351941,1075139
BC00096=141865,351941,1075139
BC00097=141865,351941,1075139
BC00098=141865,351941,1075139
BC00099=141865,351941,1075139
BC00100=141865,351941,1075139
BC00101=69858,384215,1075139
BC00102=70003,439901,1075139
BC00103=70003,439901,1075139
BC00104=70003,439901,1075139
BC00105=70003,439901,1075139
BC00106=70003,439901,1075139
BC00107=70003,439901,1075139
BC00108=70003,439901,1075139
BC00109=70003,439901,1075139
BC00110=70003,439901,1075139
BC00111=70003,439901,1075139
BC00112=70003,439901,1075139
BC00113=70003,439901,1075139
BC00114=70003,439901,1075139
BC00115=70002,439901,1075136
BC00116=70002,439901,1075136
BC00117=70002,439901,1075136
BC00118=70002,439901,1075136
BC00119=70002,439901,1075136
BC00120=70002,439901,1075136
BC00121=70002,439901,1075136
BC00122=70002,439901,1075136
BC00123=110188,367149,1075138
BC00124=128414,334151,1075139
BC00125=124989,244769,1075139
BC00126=124989,244769,1075139
BC00127=124989,244769,1075139
BC00128=124989,244769,1075139
BC00129=124989,244769,1075139
BC00130=124989,244769,1075139
BC00131=124989,244769,1075139
BC00132=124989,244769,1075139
BC00133=124989,244769,1075139
BC00134=124989,244769,1075139
BC00135=124989,244769,1075139
BC00136=177732,250101,1075139
BC00137=177732,250101,1075139
BC00138=177732,250101,1075139
BC00139=177732,250101,1075139
BC00140=177732,250101,1075139
BC00141=177732,250101,1075139
BC00142=177732,250101,1075139
BC00143=177732,250101,1075139
BC00144=177732,250101,1075139
BC00145=177732,250101,1075139
BC00146=177732,250101,1075139
BC00147=177732,250101,1075139
BC00148=225959,237109,1075139
BC00149=225959,237109,1075139
BC00150=225959,237109,1075139
BC00151=225959,237109,1075139
BC00152=225959,237109,1075139
BC00153=225959,237109,1075139
BC00154=225959,237109,1075139
BC00155=225959,237109,1075139
BC00156=225959,237109,1075139
BC00157=225959,237109,1075139
BC00158=225959,237109,1075139
BC00159=225959,237109,1075139
BC00160=254397,237082,1075139
BC00161=252531,235586,1075139
BC00162=252532,235590,1075139
BC00163=252567,235458,1075139
BC00164=252003,232434,1075139
BC00165=252567,235458,1075139
BC00166=252149,235322,1075139
BC00167=249014,235866,1075139
BC00168=252149,235322,1075139
BC00169=258680,240559,1075139
BC00170=251432,238461,1075139
BC00171=250535,233661,1075139
BC00172=250176,231741,1075139
BC00173=250177,231745,1075139
BC00174=250057,231714,1075139
BC00175=249493,228690,1075139
BC00176=250057,231714,1075139
BC00177=251313,238434,1075139
BC00178=248423,197074,1075139
BC00179=271622,172824,1075139
BC00180=314931,127552,1075139
BC00181=311264,133736,1075139
BC00182=310393,135204,1075139
BC00183=310393,135208,1075139
BC00184=310393,135204,1075139
BC00185=284313,123972,1075139
BC00186=285915,126627,1075139
BC00187=284313,123972,1075139
BC00188=333572,150784,1075139
BC00189=330819,152330,1075139
BC00190=333572,150784,1075139
BC00191=340444,144716,1075139
BC00192=296117,142422,1075139
BC00193=279303,141551,1075139
BC00194=281879,145825,1075139
BC00195=282910,147535,1075139
BC00196=282910,147539,1075139
BC00197=282728,147623,1075139
BC00198=284330,150278,1075139
BC00199=282728,147623,1075139
BC00200=279121,141639,1075139
BC00201=253491,161905,1074208
BC00202=222040,181387,1074524
BC00203=146318,174247,1075139
BC00204=66189,145086,1075139
BC00205=66189,145086,1075139
BC00206=66189,145086,1075139
BC00207=66189,145086,1075139
BC00208=66189,145086,1075139
BC00209=66189,145086,1075139
BC00210=66189,145086,1075139
BC00211=66189,145086,1075139
BC00212=66189,145086,1075139
BC00213=66189,145086,1075139
BC00214=66189,145086,1075139
BC00215=66189,145086,1075139
BC00216=125013,230326,1075139
BC00217=190374,217976,1075139
BC00218=190374,217976,1075139
BC00219=190374,217976,1075137
BC00220=190374,217976,1075139
BC00221=190374,217976,1075139
BC00222=190374,217976,1075139
BC00223=190374,217976,1075139
BC00224=190374,217976,1075139
BC00225=190374,217976,1075139
BC00226=190374,217976,1075139
BC00227=190374,217976,1075139
BC00228=190374,217976,1075139
BC00229=190374,217976,1075139
BC00230=103347,302074,1075139
BC00231=35288,367844,1075139
BC00232=35288,367844,1075139
BC00233=35288,367844,1075139
BC00234=35288,367844,1075139
BC00235=35288,367844,1075139
BC00236=35288,367844,1075139
BC00237=35288,367844,1075139
BC00238=35288,367844,1075139
BC00239=35288,367844,1075139
BC00240=35288,367844,1075139
BC00241=35288,367844,1075139
BC00242=35288,367844,1075139
BC00243=167951,390164,1075139
BC00244=311289,291148,1075139
BC00245=311289,291148,1075139
BC00246=311289,291148,1075139
BC00247=311289,291148,1075139
BC00248=311289,291148,1075139
BC00249=311289,291148,1075139
BC00250=311289,291148,1075139
BC00251=311289,291148,1075139
BC00252=311289,291148,1075139
BC00253=311289,291148,1075139
BC00254=311289,291148,1075139
BC00255=311289,291148,1075139
BC00256=113164,365819,1075193
BC00257=113164,365819,1075193
BC00258=113164,365819,1075193
BC00259=113164,365819,1075193
BC00260=113164,365819,1075193
BC00261=113164,365819,1075193
BC00262=113164,365819,1075193
BC00263=113164,365819,1075193
BC00264=113164,365819,1075193
BC00265=113164,365819,1075193
BC00266=113164,365819,1075193
BC00267=113164,365819,1075193
BC00268=355746,222574,1075139
BC00269=355746,222574,1075139
BC00270=355746,222574,1075139
BC00271=355746,222574,1075139
BC00272=355746,222574,1075139
BC00273=355746,222574,1075139
BC00274=355746,222574,1075139
BC00275=355746,222574,1075139
BC00276=397187,215310,1075139
BC00277=397187,215310,1075139
BC00278=397187,215310,1075139
BC00279=397187,215310,1075139
BC00280=397187,215310,1075139
BC00281=397187,215310,1075139
BC00282=397187,215310,1075139
BC00283=397187,215310,1075139
BC00284=279766,237198,1075139
BC00285=264316,222674,1075139
BC00286=264316,222674,1075139
BC00287=264316,222674,1075139
BC00288=264316,222674,1075139
BC00289=264316,222674,1075139
BC00290=264316,222674,1075139
BC00291=264316,222674,1075139
BC00292=264316,222674,1075139
BC00293=264316,222674,1075139
BC00294=264316,222674,1075139
BC00295=264316,222674,1075139
BC00296=290578,233908,1075139
BC00297=316840,245142,1075139
BC00298=316840,245142,1075139
BC00299=316840,245142,1075139
BC00300=316840,245142,1075139
BC00301=316840,245142,1075139
BC00302=316840,245142,1075139
BC00303=316840,245142,1075139
BC00304=316840,245142,1075139
BC00305=316840,245142,1075139
BC00306=316840,245142,1075139
BC00307=316840,245142,1075139
BC00308=316840,245142,1075139
BC00309=316840,245142,1075139
BC00310=316840,245142,1075139
BC00311=316840,245142,1075139
BC00312=316840,245142,1075139
BC00313=329930,299025,1075139
BC00314=337509,330221,1075139
BC00315=337509,330221,1075139
BC00316=337509,330221,1075139
BC00317=337509,330221,1075139
BC00318=337509,330221,1075139
BC00319=337509,330221,1075139
BC00320=337509,330221,1075139
BC00321=337509,330221,1075139
BC00322=238132,315732,1075139
BC00323=227190,314283,1075139
BC00324=227190,314283,1075139
BC00325=227190,314283,1075139
BC00326=227190,314283,1075139
BC00327=227190,314283,1075139
BC00328=227190,314283,1075139
BC00329=280930,302434,1075139
BC00330=280930,302434,1075139
BC00331=280930,302434,1075139
BC00332=280930,302434,1075139
BC00333=280930,302434,1075139
BC00334=280930,302434,1075139
BC00335=280930,302434,1075139
BC00336=280930,302434,1075139
BC00337=239245,340064,1075139
BC00338=207853,332755,1075139
BC00339=207853,332755,1075139
BC00340=207854,332756,1075137
BC00341=207853,332755,1075139
BC00342=207853,332755,1075139
BC00343=207853,332755,1075139
BC00344=207853,332755,1075139
BC00345=207853,332755,1075139
BC00346=207980,332259,1075139
BC00347=184516,253601,1075139
BC00348=163659,183682,1075139
BC00349=164098,188368,1075139
BC00350=164273,190242,1075139
BC00351=160175,192611,1075139
BC00352=158434,193619,1075139
BC00353=154337,195990,1075139
BC00354=154162,194116,1075139
BC00355=153723,189430,1075139
BC00356=82703,215475,1075139
BC00357=82703,215475,1075139
BC00358=82704,215475,1075136
BC00359=82704,215475,1075136
BC00360=82703,215475,1075139
BC00361=82704,215475,1075137
BC00362=82703,215475,1075139
BC00363=82703,215475,1075139
BC00364=70425,241198,1075139
BC00365=70425,241198,1075139
BC00366=70425,241198,1075139
BC00367=70425,241198,1075139
BC00368=70425,241198,1075139
BC00369=70425,241198,1075139
BC00370=182202,232259,1075139
BC00371=274981,189689,1075139
BC00372=293307,181281,1075139
BC00373=293307,181281,1075139
BC00374=293307,181281,1075139
BC00375=293307,181281,1075139
BC00376=293307,181281,1075139
BC00377=293307,181281,1075139
BC00378=337228,130480,1075139
BC00379=337228,130480,1075139
BC00380=337228,130480,1075139
BC00381=337228,130480,1075139
BC00382=337228,130480,1075139
BC00383=337228,130480,1075139
BC00384=337228,130480,1075139
BC00385=227414,207984,1075139
BC00386=114998,250424,1075139
BC00387=118851,252865,1075139
BC00388=120392,253841,1075139
BC00389=140979,242283,1075139
BC00390=182025,213741,1075139
BC00391=180830,212438,1075139
BC00392=177843,209180,1075139
BC00393=194784,205572,1075139
BC00394=244637,174025,1075139
BC00395=241495,179545,1075139
BC00396=240238,181752,1075139
BC00397=240238,181755,1075139
BC00398=241495,179547,1075139
BC00399=244637,174028,1075139
BC00400=244637,174025,1075139
BC00401=272679,156407,1075139
BC00402=285498,148353,1075139
BC00403=284735,144178,1075139
BC00404=282146,150110,1075139
BC00405=281110,152483,1075139
BC00406=207124,162094,1075139
BC00407=260813,132093,1075139
BC00408=212018,177166,1075139
BC00409=209211,177191,1075139
BC00410=202194,177255,1075139
BC00411=196597,207596,1075139
BC00412=175947,319541,1075139
BC00413=163596,386499,1075139
BC00414=152615,411577,1075139
BC00415=146076,409803,1075139
BC00416=143461,409093,1075139
BC00417=143581,409031,1075139
BC00418=143609,409017,1075139
BC00419=143730,408953,1075139
BC00420=146345,409663,1075139
BC00421=152884,411437,1075139
BC00422=152884,411437,1075139
BC00423=74068,445423,1075139
BC00424=74068,445423,1075139
BC00425=67271,510215,1075139
BC00426=67271,510215,1075139
BC00427=67271,510215,1075139
BC00428=67271,510215,1075139
BC00429=67271,510215,1075139
BC00430=67271,510215,1075139
BC00431=67271,551428,1075139
BC00432=67271,510215,1075139
BC00433=83379,495815,1075139
BC00434=102092,479087,1075139
BC00435=165542,422367,1075139
BC00436=222466,371481,1075139
BC00437=215798,369788,1075139
BC00438=213131,369110,1075139
BC00439=213131,369115,1075139
BC00440=213131,369116,1075139
BC00441=213132,369121,1075139
BC00442=215799,369798,1075139
BC00443=222467,371492,1075139
BC00444=173706,373999,1075139
BC00445=90340,378286,1075139
BC00446=89680,378535,1075139
BC00447=89416,378634,1075139
BC00448=85285,380949,1075139
BC00449=73307,387674,1075139
BC00450=69180,389995,1075139
BC00451=69444,389896,1075139
BC00452=70104,389647,1075139
BC00453=203953,322118,1075139
BC00454=200176,323472,1075139
BC00455=198665,324014,1075139
BC00456=196262,320031,1075139
BC00457=188009,306357,1075139
BC00458=185604,302375,1075139
BC00459=187115,301833,1075139
BC00460=190891,300479,1075139
BC00461=185791,355652,1075139
BC00462=185026,363928,1075139
BC00463=182804,358923,1075139
BC00464=181915,356921,1075139
BC00465=205267,343878,1075139
BC00466=246890,326475,1075139
BC00467=246890,326475,1075139
BC00468=248198,328377,1075139
BC00469=251468,333132,1075139
BC00470=176986,357038,1075139
BC00471=153547,361674,1075139
BC00472=140004,364885,1075139
BC00473=143591,358849,1075139
BC00474=145026,356434,1075139
BC00475=145026,356440,1075139
BC00476=143591,358854,1075139
BC00477=140005,364891,1075139
BC00478=140004,364885,1075139
BC00479=325284,234232,1075139
BC00480=326082,229506,1075139
BC00481=326401,227615,1075139
BC00482=373926,219365,1075139
BC00483=373607,221255,1075139
BC00484=372809,225981,1075139
BC00485=388697,345914,1075139
BC00486=388697,345914,1075139
BC00487=388697,345914,1075139
BC00488=388697,345914,1075139
BC00489=388697,345914,1075139
BC00490=392605,344549,1075139
BC00491=388828,320373,1075139
BC00492=388828,320373,1075139
BC00493=388828,320373,1075139
BC00494=388828,320373,1075139
BC00495=386499,330172,1075139
BC00496=382563,328869,1075139
BC00497=382563,328869,1075139
BC00498=398158,328024,1075139
BC00499=398158,329380,1075139
BC00500=398159,329745,1075136
BC00501=398158,329745,1075139
BC00502=398158,329745,1075139
BC00503=398158,329745,1075139
BC00504=398158,330311,1075139
BC00505=398158,336209,1075139
BC00506=335540,227987,1075139
BC00507=313077,229196,1075139
BC00508=312763,223759,1075139
BC00509=312637,221584,1075139
BC00510=317340,220768,1075139
BC00511=322580,219858,1075139
BC00512=322706,222033,1075139
BC00513=323019,227470,1075139
BC00514=275774,224856,1075139
BC00515=219080,221719,1075139
BC00516=223104,219732,1075139
BC00517=224713,218937,1075139
BC00518=220803,223606,1075139
BC00519=219194,224401,1075139
BC00520=215170,226388,1075139
BC00521=283236,215079,1075139
BC00522=343567,205055,1075139
BC00523=351302,203770,1075139
BC00524=346935,202437,1075139
BC00525=345561,202216,1075139
BC00526=346824,203276,1075139
BC00527=348071,204322,1075139
BC00528=348071,204322,1075139
BC00529=349706,205694,1075139
BC00530=349706,205694,1075139
BC00531=351337,206192,1075139
BC00532=355820,207560,1075139
BC00533=351302,203770,1075139
BC00534=322578,296019,1075139
BC00535=319254,304865,1075139
BC00536=319129,308714,1075139
BC00537=319080,310253,1075139
BC00538=319080,310253,1075139
BC00539=310142,308745,1075139
BC00540=310266,304896,1075139
BC00541=287916,292062,1075139
BC00542=289201,296567,1075139
BC00543=289713,298368,1075138
BC00544=286395,298387,1075139
BC00545=285163,296589,1075139
BC00546=283878,292083,1075139
BC00547=317870,285761,1075139
BC00548=321392,285753,1075139
BC00549=251901,275423,1075139
BC00550=191207,304894,1075139
BC00551=191207,266401,1075139
BC00552=186603,263429,1075139
BC00553=184761,262240,1075139
BC00554=132341,285564,1075139
BC00555=148443,282769,1075139
BC00556=150302,283070,1075139
BC00557=172103,286599,1075139
BC00558=172318,288256,1075139
BC00559=172855,292400,1075139
BC00560=285119,269376,1075139
BC00561=282278,265391,1075139
BC00562=278353,264835,1075139
BC00563=250826,275081,1075139
BC00564=302465,266011,1075139
BC00565=235375,264102,1075139
BC00566=233190,265674,1075139
BC00567=227726,269605,1075139
BC00568=172855,315333,1075139
BC00569=140733,366897,1075139
BC00570=114376,409206,1075139
BC00571=114376,409206,1075139
BC00572=114376,409206,1075139
BC00573=114376,409206,1075139
BC00574=114376,409206,1075139
BC00575=114376,409206,1075139
BC00576=114376,409206,1075139
BC00577=114376,409206,1075139
BC00578=147405,398473,1075139
BC00579=157458,395206,1075139
BC00580=157458,395206,1075139
BC00581=157458,395206,1075139
BC00582=157458,395206,1075139
BC00583=157458,395206,1075139
BC00584=157458,395206,1075139
BC00585=157458,395206,1075139
BC00586=157458,395206,1075139
BC00587=188960,381179,1075139
BC00588=188960,381179,1075139
BC00589=188960,381179,1075139
BC00590=188960,381179,1075139
BC00591=188960,381179,1075139
BC00592=188960,381179,1075139
BC00593=188960,381179,1075139
BC00594=188960,381179,1075139
BC00595=147625,408083,1075139
BC00596=198560,344942,1075139
BC00597=232795,256231,1075139
BC00598=232880,256766,1075139
BC00599=232019,251392,1075139
BC00600=231675,249242,1075139
BC00601=233668,248110,1075136
BC00602=218902,238549,1075139
BC00603=218471,244286,1075139
BC00604=199699,224542,1075139
BC00605=202215,218867,1075139
BC00606=203221,216597,1075139
BC00607=199754,218156,1075139
BC00608=198670,220460,1075139
BC00609=195959,226222,1075139
BC00610=268303,231304,1075139
BC00611=299756,233514,1075139
BC00612=294945,229330,1075139
BC00613=302009,223004,1075139
BC00614=302009,223004,1075139
BC00615=302846,222538,1075139
BC00616=304965,224120,1075139
BC00617=310261,228077,1075139
BC00618=299756,243306,1075139
BC00619=156352,322739,1075139
BC00620=114174,246219,1075139
BC00621=112841,242871,1075139
BC00622=112308,241531,1075139
BC00623=57422,251060,1075139
BC00624=57422,251060,1075139
BC00625=57956,252399,1075139
BC00626=59288,255747,1075139
BC00627=59943,258536,1075139
BC00628=60147,259407,1075139
BC00629=64884,255680,1075139
BC00630=66778,254190,1075139
BC00631=70910,256327,1075139
BC00632=86698,269328,1075139
BC00633=88860,273213,1075139
BC00634=87231,275075,1075139
BC00635=83158,279731,1075139
BC00636=93067,279347,1075139
BC00637=96346,273122,1075139
BC00638=97657,270632,1075139
BC00639=102091,274513,1075139
BC00640=93718,264741,1075139
BC00641=92112,266911,1075139
BC00642=88099,272337,1075139
BC00643=59288,336257,1075139
BC00644=302181,233758,1075139
BC00645=302181,233758,1075139
BC00646=297668,231154,1075139
BC00647=295863,230112,1075139
BC00648=304723,191150,1075139
BC00649=304707,211490,1075139
BC00650=296415,162637,1075139
BC00651=295280,145830,1075139
BC00652=298649,140382,1075139
BC00653=298649,140382,1075139
BC00654=21198,517278,1075139
BC00655=21198,517278,272386
BC00656=236183,512688,426384
BC00657=241698,501265,473364
BC00658=337027,399428,130104
BC00659=337027,399428,130104
BC00660=337027,399428,130104
BC00661=337027,399428,130104
BC00662=337027,399428,130104
BC00663=337027,399428,130104
BC00664=337027,399428,130104
BC00665=337027,399428,130104
BC00666=337027,399428,130104
BC00667=337027,399428,130104
BC00668=337027,399428,130104
BC00669=337027,399428,130104
BC00670=337027,399428,130104
BC00671=330275,399428,185956
BC00672=327708,399428,238931
BC00673=339066,399428,299662
BC00674=339066,399428,299662
BC00675=339066,399428,299662
BC00676=339066,399428,299662
BC00677=339066,399428,299662
BC00678=339066,399428,299662
BC00679=339066,399428,299662
BC00680=318740,399428,287557
BC00681=318740,399428,287557
BC00682=318740,399428,287557
BC00683=318740,399428,287557
BC00684=318740,399428,287557
BC00685=318740,399428,287557
BC00686=318740,399428,287556
BC00687=318740,399428,287556
BC00688=318740,399428,287557
BC00689=330162,399428,353919
BC00690=360317,399428,257125
BC00691=360317,399428,211725
BC00692=319771,399428,339211
BC00693=319771,399428,338822
BC00694=319771,399428,338822
BC00695=319771,399428,338822
BC00696=319771,399428,338822
BC00697=319771,399428,338822
BC00698=319771,399428,338822
BC00699=319771,399428,338822
BC00700=319771,399428,338822
BC00701=319771,399428,338822
BC00702=345973,399428,327214
BC00703=345973,399428,327214
BC00704=345973,399428,327214
BC00705=345973,399428,327214
BC00706=345973,399428,327214
BC00707=345973,399428,327214
BC00708=345973,399428,327214
BC00709=345973,399428,327214
BC00710=345973,399428,327214
BC00711=308609,441664,384698
BC00712=276024,478499,434832
BC00713=276024,575283,434832
BC00714=237619,521913,493918
BC00715=196144,517607,511250
BC00716=196144,517607,511250
BC00717=196144,462873,429035
BC00718=164288,424980,372117
BC00719=164288,424980,372117
BC00720=164288,424980,372117
BC00721=164288,424980,372117
BC00722=164288,424980,264583
BC00723=164288,424980,264583
BC00724=164288,424980,264583
BC00725=164288,424980,264583
BC00726=164288,424980,264583
BC00727=164288,424980,264583
BC00728=172101,411691,210952
BC00729=172101,411691,210952
BC00730=172101,411691,210952
BC00731=172101,411691,210952
BC00732=172101,411691,210952
BC00733=172101,411691,210952
BC00734=172101,411691,210952
BC00735=172101,411691,210952
BC00736=172101,411691,210952
BC00737=149049,399428,133666
BC00738=149049,399428,133666
BC00739=149049,399428,133666
BC00740=149049,399428,133666
BC00741=149049,399428,133666
BC00742=149049,399428,133666
BC00743=149049,399428,133666
BC00744=149049,399428,133666
BC00745=149049,399428,133666
BC00746=149049,399428,133666
BC00747=149049,399428,133666
BC00748=149049,399428,133666
BC00749=117497,399428,17
BC00750=117497,399428,17
BC00751=117497,399428,17
BC00752=117497,399428,17
BC00753=117497,399428,17
BC00754=117497,399428,17
BC00755=117497,399428,17
BC00756=117497,399428,17
BC00757=117497,399428,17
BC00758=117497,399428,17
BC00759=117497,399428,17
BC00760=117497,399428,17
BC00761=117497,399428,17
BC00762=190596,399428,158452
BC00763=190596,399428,158452
BC00764=190596,399428,158452
BC00765=190596,399428,158452
BC00766=190596,399428,158452
BC00767=190596,399428,158452
BC00768=184890,399428,111032
BC00769=184890,399428,111032
BC00770=184890,399428,111032
BC00771=184890,399428,111032
BC00772=184890,399428,111032
BC00773=184890,399428,111032
BC00774=181331,399428,152983
BC00775=154134,399428,218288
BC00776=154134,399428,218288
BC00777=154134,399428,218288
BC00778=154134,399428,218288
BC00779=154134,399428,218288
BC00780=154134,399428,218288
BC00781=184975,456611,315847
BC00782=196144,517607,403716
BC00783=186423,517607,403716
BC00784=327910,526966,492573
BC00785=308609,441664,357815
BC00786=309533,399428,345565
BC00787=309533,399428,345565
BC00788=309533,399428,345565
BC00789=309533,399428,345565
BC00790=309533,399428,345565
BC00791=309533,399428,345565
BC00792=321183,399428,368425
BC00793=321183,399428,368425
BC00794=321183,399428,368425
BC00795=321183,399428,368425
BC00796=321183,399428,368425
BC00797=321183,399428,368425
BC00798=321183,399428,368425
BC00799=321183,399428,368425
BC00800=335575,426691,378483
BC00801=330892,405614,346398
BC00802=329518,399428,161319
BC00803=329518,399428,161319
BC00804=329518,399428,218889
BC00805=329518,399428,218889
BC00806=329518,399428,263266
BC00807=308897,399428,229969
BC00808=308897,399428,161319
BC00809=308897,399428,161319
BC00810=308897,399428,161319
BC00811=308897,399428,161319
BC00812=308897,399428,161319
BC00813=308897,399428,161319
BC00814=308897,399428,161319
BC00815=308897,399428,161319
BC00816=308897,399428,161319
BC00817=308897,399428,161319
BC00818=308897,399428,195492
BC00819=308897,399428,216551
BC00820=310346,399428,231315
BC00821=308897,399428,235780
BC00822=308897,423839,237984
BC00823=308897,424955,188701
BC00824=308897,424955,188701
BC00825=308897,424955,188701
BC00826=308897,424955,188701
BC00827=313925,430321,284628
BC00828=326274,443447,308383
BC00829=310910,490157,464438
BC00830=300297,522422,410930
BC00831=200162,428906,279701
BC00832=168597,399428,238336
BC00833=168597,399428,238336
BC00834=168597,402615,238336
BC00835=168596,407259,238336
BC00836=168597,399428,238336
BC00837=168597,399428,238336
BC00838=187380,404529,191995
BC00839=187380,404529,191995
BC00840=187380,404529,191995
BC00841=187380,404529,191995
BC00842=187380,404529,191995
BC00843=187380,404529,191995
BC00844=186601,428906,279701
BC00845=300297,522422,410930
BC00846=300297,522422,410930
BC00847=342630,448885,314477
BC00848=326007,399428,330931
BC00849=326007,399428,330931
BC00850=326007,399428,330931
BC00851=326007,399428,330931
BC00852=326007,399428,330931
BC00853=326007,399428,330931
BC00854=316493,399428,286670
BC00855=316493,399428,286670
BC00856=316494,399429,286670
BC00857=316493,399428,286670
BC00858=316493,399428,286670
BC00859=316493,399428,286670
BC00860=314385,456607,481218
BC00861=308030,561884,547494
BC00862=300297,522422,410930
BC00863=200162,428906,279701
BC00864=186942,411017,256565
BC00865=178379,399428,241578
BC00866=178379,399428,241578
BC00867=154402,399428,241578
BC00868=154402,399428,241578
BC00869=154402,399428,241578
BC00870=157953,402650,241578
BC00871=198025,419755,161008
BC00872=198025,419755,161008
BC00873=198025,419755,161008
BC00874=198025,419755,161008
BC00875=198025,419755,161008
BC00876=198025,419755,161008
BC00877=172497,428906,279701
BC00878=300297,522422,410930
BC00879=360278,522422,531204
BC00880=363238,423016,313826
BC00881=356697,405293,272548
BC00882=356697,405293,264212
BC00883=356697,405293,264212
BC00884=356697,405293,264212
BC00885=356697,405293,264212
BC00886=321363,405293,365485
BC00887=345223,399428,356445
BC00888=345223,399428,356445
BC00889=345223,399428,356445
BC00890=345223,399428,356445
BC00891=345223,399428,356445
BC00892=345223,399428,356445
BC00893=331344,423016,374962
BC00894=341151,557738,486195
BC00895=300297,522422,410930
BC00896=175905,428906,279701
BC00897=142652,399428,138777
BC00898=142652,399428,138777
BC00899=142653,399429,138776
BC00900=142652,399428,138777
BC00901=142652,399428,138777
BC00902=142652,399428,138777
BC00903=142652,399428,138777
BC00904=142652,399428,138777
BC00905=143390,406891,197989
BC00906=170952,426801,272293
BC00907=201576,488605,280359
BC00908=200162,520546,279701
BC00909=78377,519142,1075139
EC00000=-798156,-183832
EC00001=-798153,-183835
EC00002=-798156,-183832
EC00003=-798156,-183832
EC00004=-798156,-183832
EC00005=-798156,-183832
EC00006=-798156,-183832
EC00007=-798156,-183832
EC00008=-798156,-183832
EC00009=-798156,-183832
EC00010=-798156,-183832
EC00011=-798156,-183832
EC00012=-798156,-183832
EC00013=-798156,-183832
EC00014=-798156,-183832
EC00015=-798156,-183832
EC00016=-798156,-183832
EC00017=-798156,-183832
EC00018=-798156,-183832
EC00019=-798156,-183832
EC00020=-798156,-183832
EC00021=-798156,-183832
EC00022=-798156,-183832
EC00023=-798156,-183832
EC00024=-798156,-183832
EC00025=-798156,-183832
EC00026=-798156,-183832
EC00027=-798156,-183832
EC00028=-798156,-183832
EC00029=-798156,-183832
EC00030=-798156,-183832
EC00031=-798156,-183832
EC00032=-798156,-183832
EC00033=-798156,-183832
EC00034=-798156,-183832
EC00035=-798156,-183832
EC00036=-798156,-183832
EC00037=-798156,-183832
EC00038=-798156,-183832
EC00039=-798156,-183832
EC00040=-798156,-183832
EC00041=-798156,-183832
EC00042=-798156,-183832
EC00043=-798156,-183832
EC00044=-798156,-183832
EC00045=-798156,-183832
EC00046=-798156,-183832
EC00047=-798156,-183832
EC00048=-798156,-183832
EC00049=-798156,-183832
EC00050=-798156,-183832
EC00051=-798156,-183832
EC00052=-798156,-183832
EC00053=-798156,-183832
EC00054=-798156,-183832
EC00055=-798156,-183832
EC00056=-798156,-183832
EC00057=-798156,-183832
EC00058=-798156,-183832
EC00059=-798156,-183832
EC00060=-798156,-183832
EC00061=-798156,-183832
EC00062=-798156,-183832
EC00063=-798156,-183832
EC00064=-798156,-183832
EC00065=-798156,-183832
EC00066=-798156,-183832
EC00067=-798156,-183832
EC00068=-798156,-183832
EC00069=-798156,-183832
EC00070=-798156,-183832
EC00071=-798156,-183832
EC00072=-798156,-183832
EC00073=-798156,-183832
EC00074=-798156,-183832
EC00075=-798156,-183832
EC00076=-798156,-183832
EC00077=-798156,-183832
EC00078=-798156,-183832
EC00079=-798156,-183832
EC00080=-798156,-183832
EC00081=-798156,-183832
EC00082=-798156,-183832
EC00083=-798156,-183832
EC00084=-798156,-183832
EC00085=-798156,-183832
EC00086=-798156,-183832
EC00087=-798156,-183832
EC00088=-798156,-183832
EC00089=-798156,-183832
EC00090=-798156,-183832
EC00091=-798156,-183832
EC00092=-798156,-183832
EC00093=-798156,-183832
EC00094=-798156,-183832
EC00095=-798156,-183832
EC00096=-798156,-183832
EC00097=-798156,-183832
EC00098=-798156,-183832
EC00099=-798156,-183832
EC00100=-798156,-183832
EC00101=-798156,-183832
EC00102=-798156,-183832
EC00103=-798156,-183832
EC00104=-798156,-183832
EC00105=-798156,-183832
EC00106=-798156,-183832
EC00107=-798156,-183832
EC00108=-798156,-183832
EC00109=-798156,-183832
EC00110=-798156,-183832
EC00111=-798156,-183832
EC00112=-798156,-183832
EC00113=-798156,-183832
EC00114=-798156,-183832
EC00115=-798155,-183832
EC00116=-798155,-183832
EC00117=-798155,-183832
EC00118=-798155,-183832
EC00119=-798155,-183832
EC00120=-798155,-183832
EC00121=-798155,-183832
EC00122=-798155,-183832
EC00123=-798155,-183832
EC00124=-798156,-183832
EC00125=-798156,-183832
EC00126=-798156,-183832
EC00127=-798156,-183832
EC00128=-798156,-183832
EC00129=-798156,-183832
EC00130=-798156,-183832
EC00131=-798156,-183832
EC00132=-798156,-183832
EC00133=-798156,-183832
EC00134=-798156,-183832
EC00135=-798156,-183832
EC00136=-798156,-183832
EC00137=-798156,-183832
EC00138=-798156,-183832
EC00139=-798156,-183832
EC00140=-798156,-183832
EC00141=-798156,-183832
EC00142=-798156,-183832
EC00143=-798156,-183832
EC00144=-798156,-183832
EC00145=-798156,-183832
EC00146=-798156,-183832
EC00147=-798156,-183832
EC00148=-798156,-183832
EC00149=-798156,-183832
EC00150=-798156,-183832
EC00151=-798156,-183832
EC00152=-798156,-183832
EC00153=-798156,-183832
EC00154=-798156,-183832
EC00155=-798156,-183832
EC00156=-798156,-183832
EC00157=-798156,-183832
EC00158=-798156,-183832
EC00159=-798156,-183832
EC00160=-798156,-183832
EC00161=-798156,-183832
EC00162=-798156,-183832
EC00163=-798156,-183832
EC00164=-798156,-183832
EC00165=-798156,-183832
EC00166=-798156,-183832
EC00167=-798156,-183832
EC00168=-798156,-183832
EC00169=-798156,-183832
EC00170=-798156,-183832
EC00171=-798156,-183832
EC00172=-798156,-183832
EC00173=-798156,-183832
EC00174=-798156,-183832
EC00175=-798156,-183832
EC00176=-798156,-183832
EC00177=-798156,-183832
EC00178=-798156,-183832
EC00179=-798156,-183832
EC00180=-798156,-183832
EC00181=-798156,-183832
EC00182=-798156,-183832
EC00183=-798156,-183832
EC00184=-798156,-183832
EC00185=-798156,-183832
EC00186=-798156,-183832
EC00187=-798156,-183832
EC00188=-798156,-183832
EC00189=-798156,-183832
EC00190=-798156,-183832
EC00191=-798156,-183832
EC00192=-798156,-183832
EC00193=-798156,-183832
EC00194=-798156,-183832
EC00195=-798156,-183832
EC00196=-798156,-183832
EC00197=-798156,-183832
EC00198=-798156,-183832
EC00199=-798156,-183832
EC00200=-798156,-183832
EC00201=-798156,-183832
EC00202=-798156,-183832
EC00203=-798156,-183832
EC00204=-798156,-183832
EC00205=-798156,-183832
EC00206=-798156,-183832
EC00207=-798156,-183832
EC00208=-798156,-183832
EC00209=-798156,-183832
EC00210=-798156,-183832
EC00211=-798156,-183832
EC00212=-798156,-183832
EC00213=-798156,-183832
EC00214=-798156,-183832
EC00215=-798156,-183832
EC00216=-798156,-183832
EC00217=-798156,-183832
EC00218=-798156,-183832
EC00219=-798154,-183834
EC00220=-798156,-183832
EC00221=-798156,-183832
EC00222=-798156,-183832
EC00223=-798156,-183832
EC00224=-798156,-183832
EC00225=-798156,-183832
EC00226=-798156,-183832
EC00227=-798156,-183832
EC00228=-798156,-183832
EC00229=-798156,-183832
EC00230=-798156,-183832
EC00231=-798156,-183832
EC00232=-798156,-183832
EC00233=-798156,-183832
EC00234=-798156,-183832
EC00235=-798156,-183832
EC00236=-798156,-183832
EC00237=-798156,-183832
EC00238=-798156,-183832
EC00239=-798156,-183832
EC00240=-798156,-183832
EC00241=-798156,-183832
EC00242=-798156,-183832
EC00243=-798156,-183832
EC00244=-798156,-183832
EC00245=-798156,-183832
EC00246=-798156,-183832
EC00247=-798156,-183832
EC00248=-798156,-183832
EC00249=-798156,-183832
EC00250=-798156,-183832
EC00251=-798156,-183832
EC00252=-798156,-183832
EC00253=-798156,-183832
EC00254=-798156,-183832
EC00255=-798156,-183832
EC00256=-798156,-183832
EC00257=-798156,-183832
EC00258=-798156,-183832
EC00259=-798156,-183832
EC00260=-798156,-183832
EC00261=-798156,-183832
EC00262=-798156,-183832
EC00263=-798156,-183832
EC00264=-798156,-183832
EC00265=-798156,-183832
EC00266=-798156,-183832
EC00267=-798156,-183832
EC00268=-798156,-183832
EC00269=-798156,-183832
EC00270=-798156,-183832
EC00271=-798156,-183832
EC00272=-798156,-183832
EC00273=-798156,-183832
EC00274=-798156,-183832
EC00275=-798156,-183832
EC00276=-798156,-183832
EC00277=-798156,-183832
EC00278=-798156,-183832
EC00279=-798156,-183832
EC00280=-798156,-183832
EC00281=-798156,-183832
EC00282=-798156,-183832
EC00283=-798156,-183832
EC00284=-798156,-183832
EC00285=-798156,-183832
EC00286=-798156,-183832
EC00287=-798156,-183832
EC00288=-798156,-183832
EC00289=-798156,-183832
EC00290=-798156,-183832
EC00291=-798156,-183832
EC00292=-798156,-183832
EC00293=-798156,-183832
EC00294=-798156,-183832
EC00295=-798156,-183832
EC00296=-798156,-183832
EC00297=-798156,-183832
EC00298=-798156,-183832
EC00299=-798156,-183832
EC00300=-798156,-183832
EC00301=-798156,-183832
EC00302=-798156,-183832
EC00303=-798156,-183832
EC00304=-798156,-183832
EC00305=-798156,-183832
EC00306=-798156,-183832
EC00307=-798156,-183832
EC00308=-798156,-183832
EC00309=-798156,-183832
EC00310=-798156,-183832
EC00311=-798156,-183832
EC00312=-798156,-183832
EC00313=-798156,-183832
EC00314=-798156,-183832
EC00315=-798156,-183832
EC00316=-798156,-183832
EC00317=-798156,-183832
EC00318=-798156,-183832
EC00319=-798156,-183832
EC00320=-798156,-183832
EC00321=-798156,-183832
EC00322=-798156,-183832
EC00323=-798156,-183832
EC00324=-798156,-183832
EC00325=-798156,-183832
EC00326=-798156,-183832
EC00327=-798156,-183832
EC00328=-798156,-183832
EC00329=-798156,-183832
EC00330=-798156,-183832
EC00331=-798156,-183832
EC00332=-798156,-183832
EC00333=-798156,-183832
EC00334=-798156,-183832
EC00335=-798156,-183832
EC00336=-798156,-183832
EC00337=-798156,-183832
EC00338=-798156,-183832
EC00339=-798156,-183832
EC00340=-798152,-183835
EC00341=-798156,-183832
EC00342=-798156,-183832
EC00343=-798156,-183832
EC00344=-798156,-183832
EC00345=-798156,-183832
EC00346=-798156,-183832
EC00347=-798156,-183832
EC00348=-798156,-183832
EC00349=-798156,-183832
EC00350=-798156,-183832
EC00351=-798156,-183832
EC00352=-798156,-183832
EC00353=-798156,-183832
EC00354=-798156,-183832
EC00355=-798156,-183832
EC00356=-798156,-183832
EC00357=-798156,-183832
EC00358=-798155,-183832
EC00359=-798155,-183832
EC00360=-798156,-183832
EC00361=-798155,-183832
EC00362=-798156,-183832
EC00363=-798156,-183832
EC00364=-798156,-183832
EC00365=-798156,-183832
EC00366=-798156,-183832
EC00367=-798156,-183832
EC00368=-798156,-183832
EC00369=-798156,-183832
EC00370=-798156,-183832
EC00371=-798156,-183832
EC00372=-798156,-183832
EC00373=-798156,-183832
EC00374=-798156,-183832
EC00375=-798156,-183832
EC00376=-798156,-183832
EC00377=-798156,-183832
EC00378=-798156,-183832
EC00379=-798156,-183832
EC00380=-798156,-183832
EC00381=-798156,-183832
EC00382=-798156,-183832
EC00383=-798156,-183832
EC00384=-798156,-183832
EC00385=-798156,-183832
EC00386=-798156,-183832
EC00387=-798156,-183832
EC00388=-798156,-183832
EC00389=-798156,-183832
EC00390=-798156,-183832
EC00391=-798156,-183832
EC00392=-798156,-183832
EC00393=-798156,-183832
EC00394=-798156,-183832
EC00395=-798156,-183832
EC00396=-798156,-183832
EC00397=-798156,-183832
EC00398=-798156,-183832
EC00399=-798156,-183832
EC00400=-798156,-183832
EC00401=-798156,-183832
EC00402=-798156,-183832
EC00403=-798156,-183832
EC00404=-798156,-183832
EC00405=-798156,-183832
EC00406=-798156,-183832
EC00407=-798156,-183832
EC00408=-798156,-183832
EC00409=-798156,-183832
EC00410=-798156,-183832
EC00411=-798156,-183832
EC00412=-798156,-183832
EC00413=-798156,-183832
EC00414=-798156,-183832
EC00415=-798156,-183832
EC00416=-798156,-183832
EC00417=-798156,-183832
EC00418=-798156,-183832
EC00419=-798156,-183832
EC00420=-798156,-183832
EC00421=-798156,-183832
EC00422=-798156,-183832
EC00423=-798156,-183832
EC00424=-798156,-183832
EC00425=-798156,-183832
EC00426=-798156,-183832
EC00427=-798156,-183832
EC00428=-798156,-183832
EC00429=-798156,-183832
EC00430=-798156,-183832
EC00431=-798156,-183832
EC00432=-798156,-183832
EC00433=-798156,-183832
EC00434=-798156,-183832
EC00435=-798156,-183832
EC00436=-798156,-183832
EC00437=-798156,-183832
EC00438=-798156,-183832
EC00439=-798156,-183832
EC00440=-798156,-183832
EC00441=-798156,-183832
EC00442=-798156,-183832
EC00443=-798156,-183832
EC00444=-798156,-183832
EC00445=-798156,-183832
EC00446=-798156,-183832
EC00447=-798156,-183832
EC00448=-798156,-183832
EC00449=-798156,-183832
EC00450=-798156,-183832
EC00451=-798156,-183832
EC00452=-798156,-183832
EC00453=-798156,-183832
EC00454=-798156,-183832
EC00455=-798156,-183832
EC00456=-798156,-183832
EC00457=-798156,-183832
EC00458=-798156,-183832
EC00459=-798156,-183832
EC00460=-798156,-183832
EC00461=-798156,-183832
EC00462=-798156,-183832
EC00463=-798156,-183832
EC00464=-798156,-183832
EC00465=-798156,-183832
EC00466=-798156,-183832
EC00467=-798156,-183832
EC00468=-798156,-183832
EC00469=-798156,-183832
EC00470=-798156,-183832
EC00471=-798156,-183832
EC00472=-798156,-183832
EC00473=-798156,-183832
EC00474=-798156,-183832
EC00475=-798156,-183832
EC00476=-798156,-183832
EC00477=-798156,-183832
EC00478=-798156,-183832
EC00479=-798156,-183832
EC00480=-798156,-183832
EC00481=-798156,-183832
EC00482=-798156,-183832
EC00483=-798156,-183832
EC00484=-798156,-183832
EC00485=-798156,-183832
EC00486=-798156,-183832
EC00487=-798156,-183832
EC00488=-798156,-183832
EC00489=-798156,-183832
EC00490=-798156,-183832
EC00491=-798156,-183832
EC00492=-798156,-183832
EC00493=-798156,-183832
EC00494=-798156,-183832
EC00495=-798156,-183832
EC00496=-798156,-183832
EC00497=-798156,-183832
EC00498=-798156,-183832
EC00499=-798156,-183832
EC00500=-798156,-183833
EC00501=-798156,-183832
EC00502=-798156,-183832
EC00503=-798156,-183832
EC00504=-798156,-183832
EC00505=-798156,-183832
EC00506=-798156,-183832
EC00507=-798156,-183832
EC00508=-798156,-183832
EC00509=-798156,-183832
EC00510=-798156,-183832
EC00511=-798156,-183832
EC00512=-798156,-183832
EC00513=-798156,-183832
EC00514=-798156,-183832
EC00515=-798156,-183832
EC00516=-798156,-183832
EC00517=-798156,-183832
EC00518=-798156,-183832
EC00519=-798156,-183832
EC00520=-798156,-183832
EC00521=-798156,-183832
EC00522=-798156,-183832
EC00523=-798156,-183832
EC00524=-798156,-183832
EC00525=-798156,-183832
EC00526=-798156,-183832
EC00527=-798156,-183832
EC00528=-798156,-183832
EC00529=-798156,-183832
EC00530=-798156,-183832
EC00531=-798156,-183832
EC00532=-798156,-183832
EC00533=-798156,-183832
EC00534=-798156,-183832
EC00535=-798156,-183832
EC00536=-798156,-183832
EC00537=-798156,-183832
EC00538=-798156,-183832
EC00539=-798156,-183832
EC00540=-798156,-183832
EC00541=-798156,-183832
EC00542=-798156,-183832
EC00543=-798155,-183835
EC00544=-798155,-183836
EC00545=-798156,-183832
EC00546=-798156,-183832
EC00547=-798156,-183832
EC00548=-798156,-183832
EC00549=-798156,-183832
EC00550=-798156,-183832
EC00551=-798156,-183832
EC00552=-798156,-183832
EC00553=-798156,-183832
EC00554=-798156,-183832
EC00555=-798156,-183832
EC00556=-798156,-183832
EC00557=-798156,-183832
EC00558=-798156,-183832
EC00559=-798156,-183832
EC00560=-798156,-183832
EC00561=-798156,-183832
EC00562=-798156,-183832
EC00563=-798156,-183832
EC00564=-798156,-183832
EC00565=-798156,-183832
EC00566=-798156,-183832
EC00567=-798156,-183832
EC00568=-798156,-183832
EC00569=-798156,-183832
EC00570=-798156,-183832
EC00571=-798156,-183832
EC00572=-798156,-183832
EC00573=-798156,-183832
EC00574=-798156,-183832
EC00575=-798156,-183832
EC00576=-798156,-183832
EC00577=-798156,-183832
EC00578=-798156,-183832
EC00579=-798156,-183832
EC00580=-798156,-183832
EC00581=-798156,-183832
EC00582=-798156,-183832
EC00583=-798156,-183832
EC00584=-798156,-183832
EC00585=-798156,-183832
EC00586=-798156,-183832
EC00587=-798156,-183832
EC00588=-798156,-183832
EC00589=-798156,-183832
EC00590=-798156,-183832
EC00591=-798156,-183832
EC00592=-798156,-183832
EC00593=-798156,-183832
EC00594=-798156,-183832
EC00595=-798156,-183832
EC00596=-798156,-183832
EC00597=-798156,-183832
EC00598=-798156,-183832
EC00599=-798156,-183832
EC00600=-798156,-183832
EC00601=-798155,-183832
EC00602=-798156,-183832
EC00603=-798156,-183832
EC00604=-798156,-183832
EC00605=-798156,-183832
EC00606=-798156,-183832
EC00607=-798156,-183832
EC00608=-798156,-183832
EC00609=-798156,-183832
EC00610=-798156,-183832
EC00611=-798156,-183832
EC00612=-798156,-183832
EC00613=-798156,-183832
EC00614=-798156,-183832
EC00615=-798156,-183832
EC00616=-798156,-183832
EC00617=-798156,-183832
EC00618=-798156,-183832
EC00619=-798156,-183832
EC00620=-798156,-183832
EC00621=-798156,-183832
EC00622=-798156,-183832
EC00623=-798156,-183832
EC00624=-798156,-183832
EC00625=-798156,-183832
EC00626=-798156,-183832
EC00627=-798156,-183832
EC00628=-798156,-183832
EC00629=-798156,-183832
EC00630=-798156,-183832
EC00631=-798156,-183832
EC00632=-798156,-183832
EC00633=-798156,-183832
EC00634=-798156,-183832
EC00635=-798156,-183832
EC00636=-798156,-183832
EC00637=-798156,-183832
EC00638=-798156,-183832
EC00639=-798156,-183832
EC00640=-798156,-183832
EC00641=-798156,-183832
EC00642=-798156,-183832
EC00643=-798156,-183832
EC00644=-798156,-183832
EC00645=-798156,-183832
EC00646=-798156,-183832
EC00647=-798156,-183832
EC00648=-798156,-183832
EC00649=-798156,-183832
EC00650=-798156,-183832
EC00651=-798156,-183832
EC00652=-798156,-183832
EC00653=-798156,-183832
EC00654=-798156,-183832
EC00655=-798156,-183832
EC00656=-798156,-183832
EC00657=-798156,-183832
EC00658=-798156,-183832
EC00659=-798156,-183832
EC00660=-798156,-183832
EC00661=-798156,-183832
EC00662=-798156,-183832
EC00663=-798156,-183832
EC00664=-798156,-183832
EC00665=-798156,-183832
EC00666=-798156,-183832
EC00667=-798156,-183832
EC00668=-798156,-183832
EC00669=-798156,-183832
EC00670=-798156,-183832
EC00671=-798156,-183832
EC00672=-798156,-183832
EC00673=-798156,-183832
EC00674=-798156,-183832
EC00675=-798156,-183832
EC00676=-798156,-183832
EC00677=-798156,-183832
EC00678=-798156,-183832
EC00679=-798156,-183832
EC00680=-798156,-183832
EC00681=-798156,-183832
EC00682=-798156,-183832
EC00683=-798156,-183832
EC00684=-798156,-183832
EC00685=-798156,-183832
EC00686=-798154,-183833
EC00687=-798154,-183833
EC00688=-798156,-183832
EC00689=-798156,-183832
EC00690=-798156,-183832
EC00691=-798156,-183832
EC00692=-798156,-183832
EC00693=-798156,-183832
EC00694=-798156,-183832
EC00695=-798156,-183832
EC00696=-798156,-183832
EC00697=-798156,-183832
EC00698=-798156,-183832
EC00699=-798156,-183832
EC00700=-798156,-183832
EC00701=-798156,-183832
EC00702=-798156,-183832
EC00703=-798156,-183832
EC00704=-798156,-183832
EC00705=-798156,-183832
EC00706=-798156,-183832
EC00707=-798156,-183832
EC00708=-798156,-183832
EC00709=-798156,-183832
EC00710=-798156,-183832
EC00711=-798156,-183832
EC00712=-798156,-183832
EC00713=-798156,-183832
EC00714=-798156,-183832
EC00715=-798156,-183832
EC00716=-798156,-183832
EC00717=-798156,-183832
EC00718=-798156,-183832
EC00719=-798156,-183832
EC00720=-798156,-183832
EC00721=-798156,-183832
EC00722=-798156,-183832
EC00723=-798156,-183832
EC00724=-798156,-183832
EC00725=-798156,-183832
EC00726=-798156,-183832
EC00727=-798156,-183832
EC00728=-798156,-183832
EC00729=-798156,-183832
EC00730=-798156,-183832
EC00731=-798156,-183832
EC00732=-798156,-183832
EC00733=-798156,-183832
EC00734=-798156,-183832
EC00735=-798156,-183832
EC00736=-798156,-183832
EC00737=-798156,-183832
EC00738=-798156,-183832
EC00739=-798156,-183832
EC00740=-798156,-183832
EC00741=-798156,-183832
EC00742=-798156,-183832
EC00743=-798156,-183832
EC00744=-798156,-183832
EC00745=-798156,-183832
EC00746=-798156,-183832
EC00747=-798156,-183832
EC00748=-798156,-183832
EC00749=-798156,-183832
EC00750=-798156,-183832
EC00751=-798156,-183832
EC00752=-798156,-183832
EC00753=-798156,-183832
EC00754=-798156,-183832
EC00755=-798156,-183832
EC00756=-798156,-183832
EC00757=-798156,-183832
EC00758=-798156,-183832
EC00759=-798156,-183832
EC00760=-798156,-183832
EC00761=-798156,-183832
EC00762=-798156,-183832
EC00763=-798156,-183832
EC00764=-798156,-183832
EC00765=-798156,-183832
EC00766=-798156,-183832
EC00767=-798156,-183832
EC00768=-798156,-183832
EC00769=-798156,-183832
EC00770=-798156,-183832
EC00771=-798156,-183832
EC00772=-798156,-183832
EC00773=-798156,-183832
EC00774=-798156,-183832
EC00775=-798156,-183832
EC00776=-798156,-183832
EC00777=-798156,-183832
EC00778=-798156,-183832
EC00779=-798156,-183832
EC00780=-798156,-183832
EC00781=-798156,-183832
EC00782=-798156,-183832
EC00783=-798156,-183832
EC00784=-798156,-183832
EC00785=-798156,-183832
EC00786=-798156,-183832
EC00787=-798156,-183832
EC00788=-798156,-183832
EC00789=-798156,-183832
EC00790=-798156,-183832
EC00791=-798156,-183832
EC00792=-798156,-183832
EC00793=-798156,-183832
EC00794=-798156,-183832
EC00795=-798156,-183832
EC00796=-798156,-183832
EC00797=-798156,-183832
EC00798=-798156,-183832
EC00799=-798156,-183832
EC00800=-798156,-183832
EC00801=-798156,-183832
EC00802=-798156,-183832
EC00803=-798156,-183832
EC00804=-798156,-183832
EC00805=-798156,-183832
EC00806=-798156,-183832
EC00807=-798156,-183832
EC00808=-798156,-183832
EC00809=-798156,-183832
EC00810=-798156,-183832
EC00811=-798156,-183832
EC00812=-798156,-183832
EC00813=-798156,-183832
EC00814=-798156,-183832
EC00815=-798156,-183832
EC00816=-798156,-183832
EC00817=-798156,-183832
EC00818=-798156,-183832
EC00819=-798156,-183832
EC00820=-798156,-183832
EC00821=-798156,-183832
EC00822=-798156,-183832
EC00823=-798156,-183832
EC00824=-798156,-183832
EC00825=-798156,-183832
EC00826=-798156,-183832
EC00827=-798156,-183832
EC00828=-798156,-183832
EC00829=-798156,-183832
EC00830=-798156,-183832
EC00831=-798156,-183832
EC00832=-798156,-183832
EC00833=-798156,-183832
EC00834=-798156,-183832
EC00835=-798156,-183832
EC00836=-798156,-183832
EC00837=-798156,-183832
EC00838=-798156,-183832
EC00839=-798156,-183832
EC00840=-798156,-183832
EC00841=-798156,-183832
EC00842=-798156,-183832
EC00843=-798156,-183832
EC00844=-798156,-183832
EC00845=-798156,-183832
EC00846=-798156,-183832
EC00847=-798156,-183832
EC00848=-798156,-183832
EC00849=-798156,-183832
EC00850=-798156,-183832
EC00851=-798156,-183832
EC00852=-798156,-183832
EC00853=-798156,-183832
EC00854=-798156,-183832
EC00855=-798156,-183832
EC00856=-798155,-183833
EC00857=-798156,-183832
EC00858=-798156,-183832
EC00859=-798156,-183832
EC00860=-798156,-183832
EC00861=-798156,-183832
EC00862=-798156,-183832
EC00863=-798156,-183832
EC00864=-798156,-183832
EC00865=-798156,-183832
EC00866=-798156,-183832
EC00867=-798156,-183832
EC00868=-798156,-183832
EC00869=-798156,-183832
EC00870=-798156,-183832
EC00871=-798156,-183832
EC00872=-798156,-183832
EC00873=-798156,-183832
EC00874=-798156,-183832
EC00875=-798156,-183832
EC00876=-798156,-183832
EC00877=-798156,-183832
EC00878=-798156,-183832
EC00879=-798156,-183832
EC00880=-798156,-183832
EC00881=-798156,-183832
EC00882=-798156,-183832
EC00883=-798156,-183832
EC00884=-798156,-183832
EC00885=-798156,-183832
EC00886=-798156,-183832
EC00887=-798156,-183832
EC00888=-798156,-183832
EC00889=-798156,-183832
EC00890=-798156,-183832
EC00891=-798156,-183832
EC00892=-798156,-183832
EC00893=-798156,-183832
EC00894=-798156,-183832
EC00895=-798156,-183832
EC00896=-798156,-183832
EC00897=-798156,-183832
EC00898=-798156,-183832
EC00899=-798155,-183834
EC00900=-798156,-183833
EC00901=-798156,-183832
EC00902=-798156,-183832
EC00903=-798156,-183832
EC00904=-798156,-183832
EC00905=-798156,-183832
EC00906=-798156,-183832
EC00907=-798156,-183832
EC00908=-798156,-183832
EC00909=-798156,-183832
///POSTYPE BASE
///RECTAN
///RCONF 0,0,0,0,1,0,0,0,0,0,0,0,0,0,0,0,0,0,0,0,0,0,0,0
P00006=2.006,1.622,-0.565,0.0000,0.0000,0.0000
P00021=0.073,2.058,-0.109,0.0000,0.0000,0.0000
P00022=2.006,1.622,-0.565,0.0000,0.0000,0.0000
///RCONF 0,0,0,0,0,0,0,0,0,0,0,0,0,0,0,0,0,0,0,0,0,0,0,0
P00023=-2.957,-4.083,2.762,0.0000,0.0000,0.0000
P00024=-1.466,-0.226,-0.419,0.0000,0.0000,0.0000
P00025=3.643,0.007,-2.585,0.0000,0.0000,0.0000
P00026=2.644,0.055,-2.583,0.0000,0.0000,0.0000
P00027=2.278,0.099,-4.210,0.0000,0.0000,0.0000
P00028=-1.778,-0.182,-2.050,0.0000,0.0000,0.0000
P00029=1.749,4.006,-0.261,0.0000,0.0000,0.0000
P00030=-0.014,-0.768,0.131,0.0000,0.0000,0.0000
P00031=-0.170,0.039,-0.647,0.0000,0.0000,0.0000
P00032=-0.423,0.157,3.222,0.0000,0.0000,0.0000
P00033=0.854,-1.099,3.047,0.0000,0.0000,0.0000
///RCONF 0,0,0,0,1,0,0,0,0,0,0,0,0,0,0,0,0,0,0,0,0,0,0,0
P00034=-8.151,9.743,-4.393,0.0000,0.0000,0.0000
///RCONF 0,0,0,0,0,0,0,0,0,0,0,0,0,0,0,0,0,0,0,0,0,0,0,0
P00035=0.390,-0.027,1.040,0.0000,0.0000,0.0000
P00040=2.716,-0.016,3.014,0.0000,0.0000,0.0000
P00041=-0.109,0.014,0.966,0.0000,0.0000,0.0000
P00042=-0.220,0.371,-0.613,0.0000,0.0000,0.0000
P00043=-0.179,-5.890,-3.227,0.0000,0.0000,0.0000
P00044=-8.560,-7.557,-5.232,0.0000,0.0000,0.0000
P00045=-8.836,-6.632,-1.438,0.0000,0.0000,0.0000
P00046=-7.725,-0.107,-2.878,0.0000,0.0000,0.0000
///RCONF 0,1,0,0,0,0,0,0,0,0,0,0,0,0,0,0,0,0,0,0,0,0,0,0
P00047=0.052,4.745,-6.175,0.0000,0.0000,0.0000
///RCONF 0,0,0,0,0,0,0,0,0,0,0,0,0,0,0,0,0,0,0,0,0,0,0,0
P00048=-10.315,0.035,-3.101,0.0000,0.0000,0.0000
P00049=-9.638,1.690,-2.627,0.0000,0.0000,0.0000
P00050=-0.123,2.174,-1.314,0.0000,0.0000,0.0000
P00051=-5.945,4.696,-10.293,0.0000,0.0000,0.0000
P00052=-0.153,5.586,-7.982,0.0000,0.0000,0.0000
P00053=0.015,-0.644,-4.942,0.0000,0.0000,0.0000
P00054=-0.184,15.039,-0.270,0.0000,0.0000,0.0000
P00061=1211.499,975.999,-261.374,0.5148,35.2356,175.5099
P00062=1205.574,689.500,-262.704,0.5159,35.2461,175.5270
P00063=1197.217,207.358,-268.729,0.4863,35.2395,175.4586
P00069=2.618,0.069,-17.797,0.0000,0.0000,0.0000
P00071=-2.048,-0.034,-9.092,0.0000,0.0000,0.0000
P00072=-1.595,-0.049,-6.373,0.0000,0.0000,0.0000
P00073=-8.474,-10.331,-11.894,0.0000,0.0000,0.0000
P00074=1.731,-3.007,-10.460,0.0000,0.0000,0.0000
P00095=-11.943,-14.820,-6.815,0.0000,0.0000,0.0000
P00096=-4.844,-19.262,-10.890,0.0000,0.0000,0.0000
//INST
///DATE 2024/12/02 15:02
///ATTR SC,RW
///GROUP1 RB1,BS1
///GROUP2 ST1
NOP
'X2_8A-21A(90,0)
MOVJ C00000 BC00000 VJ=100.00  +MOVJ EC00000 VJ=100.00
CALL JOB:CLEAN-R1_KM_NEW
MOVJ C00001 BC00001 VJ=100.00  +MOVJ EC00001 VJ=100.00
MOVJ C00002 BC00002 VJ=100.00  +MOVJ EC00002 VJ=100.00
'Path S3463
SFTOF3D
MOVJ C00003 BC00003 VJ=100.00  +MOVJ EC00003 VJ=100.00
MOVL C00004 BC00004 V=666.7  +MOVJ EC00004 VJ=100.00
SMOVL C00005 BC00005 V=166.7  +MOVJ EC00005
SREFP 3 C00006 BC00006  +REFP EC00006
CALL JOB:SEARCH-R1-S13D
SET P095 P006
SFTON3D P095
SMOVL C00007 BC00007 V=166.7  +MOVJ EC00007
SMOVL C00008 BC00008 V=166.7  +MOVJ EC00008
SREFP 3 C00009 BC00009  +REFP EC00009
CALL JOB:SEARCH-R1-S13D
SET P095 P006
SFTON3D P095
SMOVL C00010 BC00010 V=166.7  +MOVJ EC00010
MOVL C00011 BC00011 V=1000.0  +MOVJ EC00011 VJ=100.00
'EndPath S3463
'Path S3464
SFTOF3D
MOVJ C00012 BC00012 VJ=100.00  +MOVJ EC00012 VJ=100.00
MOVL C00013 BC00013 V=666.7  +MOVJ EC00013 VJ=100.00
SMOVL C00014 BC00014 V=166.7  +MOVJ EC00014
SREFP 3 C00015 BC00015  +REFP EC00015
CALL JOB:SEARCH-R1-S13D
SET P096 P006
SFTON3D P096
SMOVL C00016 BC00016 V=166.7  +MOVJ EC00016
SREFP 3 C00017 BC00017  +REFP EC00017
CALL JOB:SEARCH-R1-S13D
SET P096 P006
SFTON3D P096
SMOVL C00018 BC00018 V=166.7  +MOVJ EC00018
MOVL C00019 BC00019 V=1000.0  +MOVJ EC00019 VJ=100.00
'EndPath S3464
'Path S3465
SFTOF3D
MOVJ C00020 BC00020 VJ=100.00  +MOVJ EC00020 VJ=100.00
MOVL C00021 BC00021 V=666.7  +MOVJ EC00021 VJ=100.00
SMOVL C00022 BC00022 V=166.7  +MOVJ EC00022
SREFP 3 C00023 BC00023  +REFP EC00023
CALL JOB:SEARCH-R1-S13D
SET P021 P006
SFTON3D P021
SMOVL C00024 BC00024 V=166.7  +MOVJ EC00024
SMOVL C00025 BC00025 V=166.7  +MOVJ EC00025
SREFP 3 C00026 BC00026  +REFP EC00026
CALL JOB:SEARCH-R1-S13D
SET P021 P006
SFTON3D P021
SMOVL C00027 BC00027 V=166.7  +MOVJ EC00027
MOVL C00028 BC00028 V=1000.0  +MOVJ EC00028 VJ=100.00
'EndPath S3465
'Path S3464
SFTOF3D
MOVJ C00029 BC00029 VJ=100.00  +MOVJ EC00029 VJ=100.00
MOVL C00030 BC00030 V=666.7  +MOVJ EC00030 VJ=100.00
SMOVL C00031 BC00031 V=166.7  +MOVJ EC00031
SREFP 3 C00032 BC00032  +REFP EC00032
CALL JOB:SEARCH-R1-S13D
SET P022 P006
SFTON3D P022
SMOVL C00033 BC00033 V=166.7  +MOVJ EC00033
SREFP 3 C00034 BC00034  +REFP EC00034
CALL JOB:SEARCH-R1-S13D
SET P022 P006
SFTON3D P022
SMOVL C00035 BC00035 V=166.7  +MOVJ EC00035
MOVL C00036 BC00036 V=1000.0  +MOVJ EC00036 VJ=100.00
'EndPath S3464
MOVJ C00037 BC00037 VJ=100.00  +MOVJ EC00037 VJ=100.00
'Path S3465
SFTOF3D
MOVJ C00038 BC00038 VJ=100.00  +MOVJ EC00038 VJ=100.00
MOVL C00039 BC00039 V=666.7  +MOVJ EC00039 VJ=100.00
SMOVL C00040 BC00040 V=166.7  +MOVJ EC00040
SREFP 3 C00041 BC00041  +REFP EC00041
CALL JOB:SEARCH-R1-S13D
SET P050 P006
SFTON3D P050
SMOVL C00042 BC00042 V=166.7  +MOVJ EC00042
SREFP 3 C00043 BC00043  +REFP EC00043
CALL JOB:SEARCH-R1-S13D
SET P050 P006
SFTON3D P050
SMOVL C00044 BC00044 V=166.7  +MOVJ EC00044
SMOVL C00045 BC00045 V=166.7  +MOVJ EC00045
SREFP 3 C00046 BC00046  +REFP EC00046
CALL JOB:SEARCH-R1-S13D
SET P050 P006
SFTON3D P050
SMOVL C00047 BC00047 V=166.7  +MOVJ EC00047
MOVL C00048 BC00048 V=1000.0  +MOVJ EC00048 VJ=100.00
'EndPath S3465
'Path S3466
SFTOF3D
MOVJ C00049 BC00049 VJ=100.00  +MOVJ EC00049 VJ=100.00
MOVL C00050 BC00050 V=666.7  +MOVJ EC00050 VJ=100.00
SMOVL C00051 BC00051 V=166.7  +MOVJ EC00051
SREFP 3 C00052 BC00052  +REFP EC00052
CALL JOB:SEARCH-R1-S13D
SET P051 P006
SFTON3D P051
SMOVL C00053 BC00053 V=166.7  +MOVJ EC00053
SREFP 3 C00054 BC00054  +REFP EC00054
CALL JOB:SEARCH-R1-S13D
SET P051 P006
SFTON3D P051
SMOVL C00055 BC00055 V=166.7  +MOVJ EC00055
SMOVL C00056 BC00056 V=250.0  +MOVJ EC00056
SREFP 3 C00057 BC00057  +REFP EC00057
CALL JOB:SEARCH-R1-S13D
SET P051 P006
SFTON3D P051
SMOVL C00058 BC00058 V=166.7  +MOVJ EC00058
MOVL C00059 BC00059 V=1000.0  +MOVJ EC00059 VJ=100.00
'EndPath S3466
MOVJ C00060 BC00060 VJ=100.00  +MOVJ EC00060 VJ=100.00
MOVJ C00061 BC00061 VJ=100.00  +MOVJ EC00061 VJ=100.00
'Path S3467
SFTOF3D
MOVJ C00062 BC00062 VJ=100.00  +MOVJ EC00062 VJ=100.00
MOVL C00063 BC00063 V=666.7  +MOVJ EC00063 VJ=100.00
SMOVL C00064 BC00064 V=166.7  +MOVJ EC00064
SREFP 3 C00065 BC00065  +REFP EC00065
CALL JOB:SEARCH-R1-S13D
SET P054 P006
SFTON3D P054
SMOVL C00066 BC00066 V=250.0  +MOVJ EC00066
SMOVL C00067 BC00067 V=166.7  +MOVJ EC00067
SREFP 3 C00068 BC00068  +REFP EC00068
CALL JOB:SEARCH-R1-S13D
SET P054 P006
SFTON3D P054
SMOVL C00069 BC00069 V=166.7  +MOVJ EC00069
SMOVL C00070 BC00070 V=800.0  +MOVJ EC00070
SMOVL C00071 BC00071 V=166.7  +MOVJ EC00071
SREFP 3 C00072 BC00072  +REFP EC00072
CALL JOB:SEARCH-R1-S13D
SET P054 P006
SFTON3D P054
SMOVL C00073 BC00073 V=166.7  +MOVJ EC00073
MOVL C00074 BC00074 V=1000.0  +MOVJ EC00074 VJ=100.00
'EndPath S3467
'Path S3475
SFTOF3D
MOVJ C00075 BC00075 VJ=100.00  +MOVJ EC00075 VJ=100.00
MOVL C00076 BC00076 V=666.7  +MOVJ EC00076 VJ=100.00
SMOVL C00077 BC00077 V=166.7  +MOVJ EC00077
SREFP 3 C00078 BC00078  +REFP EC00078
CALL JOB:SEARCH-R1-S13D
SET P034 P006
SFTON3D P034
SMOVL C00079 BC00079 V=166.7  +MOVJ EC00079
SMOVL C00080 BC00080 V=333.3  +MOVJ EC00080
SMOVL C00081 BC00081 V=166.7  +MOVJ EC00081
SREFP 3 C00082 BC00082  +REFP EC00082
CALL JOB:SEARCH-R1-S13D
SET P034 P006
SFTON3D P034
SMOVL C00083 BC00083 V=166.7  +MOVJ EC00083
SMOVL C00084 BC00084 V=166.7  +MOVJ EC00084
SREFP 3 C00085 BC00085  +REFP EC00085
CALL JOB:SEARCH-R1-S13D
SET P034 P006
SFTON3D P034
SMOVL C00086 BC00086 V=166.7  +MOVJ EC00086
MOVL C00087 BC00087 V=1000.0  +MOVJ EC00087 VJ=100.00
'EndPath S3475
'Path S3464
SFTOF3D
MOVJ C00088 BC00088 VJ=100.00  +MOVJ EC00088 VJ=100.00
MOVL C00089 BC00089 V=666.7  +MOVJ EC00089 VJ=100.00
SMOVL C00090 BC00090 V=166.7  +MOVJ EC00090
